KUKA KRL program: EPS_2_25990_SANMH02_A_20260122125454.src

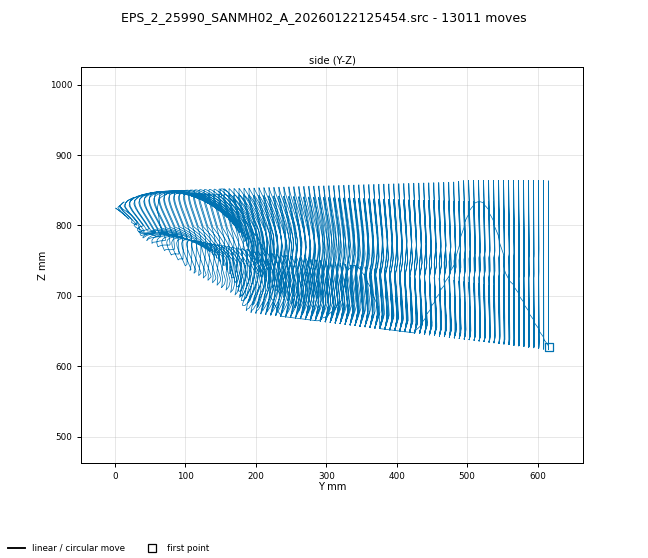
[picture p0: tool path of EPS_2_25990_SANMH02_A_20260122125454.src, 13011 of 13013 moves have a stored position in this frame; points joined in program order, loops and branches not executed]
&ACCESS RVP
&REL 4
&COMMENT QRS 19112012
&PARAM EDITMASK = *
DEF PART()
EXT BAS (BAS_COMMAND :IN,REAL :IN )
INT I
BAS (#INITMOV,0 )

;KUKA QRS Post kuka4.cps  Date:22-06-2017 !

File_ID=3005

QRS_PRE_INIT()

;Init var - Until changes are made in qrs_pre_init
Outlet_Square_prg=0
Inlet_1_Square_prg=0
Inlet_2_Square_prg=0
Inlet_3_Square_prg=0
Inlet_4_Square_prg=0
Inlet_5_Square_prg=0

Outlet_1={X 0.000, Y 498.690, Z 763.500, B 0.000, E1 0.000 }
Inlet_1={X 0.000, Y 500.880, Z 733.500, B 0.000, E1 131.000 }
Inlet_2={X 0.000, Y 537.160, Z 233.500, B 0.000, E1 218.000 }
Outlet_1_type=201
Inlet_1_type=201
Inlet_2_type=201
;QRS#1=Sidecore dimensions
;QRS#2=200-8" PVC SDR 35
;QRS#3=200-8" PVC SDR 35
;QRS#4=200-8" PVC SDR 35
;QRS#5=
;QRS#6=
;QRS#7=
;QRS#8=
;QRS#9=12-08 PSX
;QRS#10=12-08 PSX
;QRS#11=12-08 PSX
;QRS#12=
;QRS#13=
;QRS#14=
;QRS#15=
;QRS#16=1220x127x1143 3,75'
;QRS#17=EPS Height
;QRS#18=864
;QRS#19=*
;QRS#20= UPDATED VERSION 22-06-2017
;QRS#21=*
Outlet_Square=0100
Inlet_1_Square=0100
Inlet_2_Square=0100
Inlet_3_Square=0
Inlet_4_Square=0
Inlet_5_Square=0
Mill_Square=1
Outlet_Square_Prg=204
Inlet_1_Square_prg=204
Inlet_2_Square_prg=204

QRS_INIT()

$ADVANCE=5

; T1
PTP {E1 173.412,E2 173.412}
PTP {X 0,Y 615.492,A -85,B 0,C 180,E1 173.412,E2 173.412,E3 0,E4 0,E5 0,E6 0}
QRS_SPEED_INIT()
LIN {X 0,Y 615.492,Z 627.912,A -85,B 0,C 180,E1 173.412,E2 173.412,E3 0,E4 0,E5 0,E6 0} C_VEL
LIN {X 0,Y 615.475,Z 638.168,A -85,B 0,C 180,E1 170.801,E2 170.801} C_VEL
LIN {X 0,Y 615.49,Z 648.911,A -85,B 0,C 180,E1 168.139,E2 168.139} C_VEL
LIN {X 0,Y 615.487,Z 660.046,A -85,B 0,C 180,E1 165.451,E2 165.451} C_VEL
LIN {X 0,Y 615.476,Z 671.583,A -85,B 0,C 180,E1 162.729,E2 162.729} C_VEL
LIN {X 0,Y 615.485,Z 683.521,A -85,B 0,C 180,E1 159.967,E2 159.967} C_VEL
LIN {X 0,Y 615.487,Z 695.908,A -85,B 0,C 180,E1 157.155,E2 157.155} C_VEL
LIN {X 0,Y 615.494,Z 708.733,A -85,B 0,C 180,E1 154.285,E2 154.285} C_VEL
LIN {X 0,Y 615.476,Z 721.128,A -85,B 0,C 180,E1 151.55,E2 151.55} C_VEL
LIN {X 0,Y 615.494,Z 725.535,A -85,B 0,C 180,E1 150.606,E2 150.606} C_VEL
LIN {X 0,Y 615.488,Z 739.328,A -85,B 0,C 180,E1 150.351,E2 150.351} C_VEL
LIN {X 0,Y 615.49,Z 751.99,A -85,B 0,C 180,E1 149.977,E2 149.977} C_VEL
LIN {X 0,Y 615.476,Z 764.482,A -85,B 0,C 180,E1 149.46,E2 149.46} C_VEL
LIN {X 0,Y 615.493,Z 776.033,A -85,B 0,C 180,E1 148.838,E2 148.838} C_VEL
LIN {X 0,Y 615.5,Z 786.168,A -85,B 0,C 180,E1 148.154,E2 148.154} C_VEL
LIN {X 0,Y 615.499,Z 795.798,A -85,B 0,C 180,E1 147.349,E2 147.349} C_VEL
LIN {X 0,Y 615.496,Z 804.466,A -85,B 0,C 180,E1 146.463,E2 146.463} C_VEL
LIN {X 0,Y 615.497,Z 812.382,A -85,B 0,C 180,E1 145.468,E2 145.468} C_VEL
LIN {X 0,Y 615.496,Z 819.171,A -85,B 0,C 180,E1 144.385,E2 144.385} C_VEL
LIN {X 0,Y 615.496,Z 824.387,A -85,B 0,C 180,E1 143.319,E2 143.319} C_VEL
LIN {X 0,Y 615.497,Z 827.932,A -85,B 0,C 180,E1 142.373,E2 142.373} C_VEL
LIN {X 0,Y 615.498,Z 831.277,A -85,B 0,C 180,E1 141.096,E2 141.096} C_VEL
LIN {X 0,Y 615.495,Z 832.963,A -85,B 0,C 180,E1 139.909,E2 139.909} C_VEL
LIN {X 0,Y 615.492,Z 833.383,A -85,B 0,C 180,E1 138.904,E2 138.904} C_VEL
LIN {X 0,Y 615.498,Z 832.581,A -85,B 0,C 180,E1 137.648,E2 137.648} C_VEL
LIN {X 0,Y 615.499,Z 831.153,A -85,B 0,C 180,E1 136.756,E2 136.756} C_VEL
LIN {X 0,Y 615.496,Z 827.689,A -85,B 0,C 180,E1 135.46,E2 135.46} C_VEL
LIN {X 0,Y 615.495,Z 824.163,A -85,B 0,C 180,E1 134.539,E2 134.539} C_VEL
LIN {X 0,Y 615.497,Z 818.654,A -85,B 0,C 180,E1 133.431,E2 133.431} C_VEL
LIN {X 0,Y 615.495,Z 811.719,A -85,B 0,C 180,E1 132.352,E2 132.352} C_VEL
LIN {X 0,Y 615.494,Z 803.005,A -85,B 0,C 180,E1 131.284,E2 131.284} C_VEL
LIN {X 0,Y 615.498,Z 794.891,A -85,B 0,C 180,E1 130.476,E2 130.476} C_VEL
LIN {X 0,Y 615.497,Z 784.864,A -85,B 0,C 180,E1 129.662,E2 129.662} C_VEL
LIN {X 0,Y 615.487,Z 773.182,A -85,B 0,C 180,E1 128.904,E2 128.904} C_VEL
LIN {X 0,Y 615.479,Z 761.912,A -85,B 0,C 180,E1 128.328,E2 128.328} C_VEL
LIN {X 0,Y 615.483,Z 749.983,A -85,B 0,C 180,E1 127.866,E2 127.866} C_VEL
LIN {X 0,Y 615.496,Z 736.899,A -85,B 0,C 180,E1 127.504,E2 127.504} C_VEL
LIN {X 0,Y 615.489,Z 725.354,A -85,B 0,C 180,E1 127.289,E2 127.289} C_VEL
LIN {X 0,Y 615.49,Z 713.598,A -85,B 0,C 180,E1 124.701,E2 124.701} C_VEL
LIN {X 0,Y 615.481,Z 701.48,A -85,B 0,C 180,E1 122.007,E2 122.007} C_VEL
LIN {X 0,Y 615.493,Z 689.933,A -85,B 0,C 180,E1 119.405,E2 119.405} C_VEL
LIN {X 0,Y 615.476,Z 678.313,A -85,B 0,C 180,E1 116.743,E2 116.743} C_VEL
LIN {X 0,Y 615.488,Z 666.578,A -85,B 0,C 180,E1 114.008,E2 114.008} C_VEL
LIN {X 0,Y 615.492,Z 655.757,A -85,B 0,C 180,E1 111.431,E2 111.431} C_VEL
LIN {X 0,Y 615.48,Z 644.161,A -85,B 0,C 180,E1 108.603,E2 108.603} C_VEL
LIN {X 0,Y 615.484,Z 633.399,A -85,B 0,C 180,E1 105.905,E2 105.905} C_VEL
LIN {X 0,Y 615.488,Z 623.694,A -85,B 0,C 180,E1 103.369,E2 103.369} C_VEL
LIN {X 0,Y 615.476,Z 623.696,A -85,B 0,C 180,E1 100.527,E2 100.527} C_VEL
LIN {X 0,Y 615.484,Z 623.694,A -85,B 0,C 180,E1 97.875,E2 97.875} C_VEL
LIN {X 0,Y 615.485,Z 623.694,A -85,B 0,C 180,E1 95.241,E2 95.241} C_VEL
LIN {X 0,Y 615.477,Z 623.696,A -85,B 0,C 180,E1 92.618,E2 92.618} C_VEL
LIN {X 0,Y 615.491,Z 623.693,A -85,B 0,C 180,E1 90,E2 90} C_VEL
LIN {X 0,Y 615.477,Z 623.696,A -85,B 0,C 180,E1 87.382,E2 87.382} C_VEL
LIN {X 0,Y 615.485,Z 623.695,A -85,B 0,C 180,E1 84.758,E2 84.758} C_VEL
LIN {X 0,Y 615.488,Z 623.694,A -85,B 0,C 180,E1 82.124,E2 82.124} C_VEL
LIN {X 0,Y 615.477,Z 623.697,A -85,B 0,C 180,E1 79.473,E2 79.473} C_VEL
LIN {X 0,Y 615.497,Z 623.692,A -85,B 0,C 180,E1 76.799,E2 76.799} C_VEL
LIN {X 0,Y 615.481,Z 623.695,A -85,B 0,C 180,E1 74.094,E2 74.094} C_VEL
LIN {X 0,Y 615.477,Z 623.696,A -85,B 0,C 180,E1 71.353,E2 71.353} C_VEL
LIN {X 0,Y 615.492,Z 623.693,A -85,B 0,C 180,E1 68.568,E2 68.568} C_VEL
LIN {X 0,Y 615.489,Z 623.695,A -85,B 0,C 180,E1 65.728,E2 65.728} C_VEL
LIN {X 0,Y 615.482,Z 623.695,A -85,B 0,C 180,E1 63.237,E2 63.237} C_VEL
LIN {X 0,Y 615.484,Z 636.143,A -85,B 0,C 180,E1 62.823,E2 62.823} C_VEL
LIN {X 0,Y 615.481,Z 648.35,A -85,B 0,C 180,E1 62.269,E2 62.269} C_VEL
LIN {X 0,Y 615.492,Z 659.541,A -85,B 0,C 180,E1 61.615,E2 61.615} C_VEL
LIN {X 0,Y 615.5,Z 669.72,A -85,B 0,C 180,E1 60.875,E2 60.875} C_VEL
LIN {X 0,Y 615.498,Z 679.215,A -85,B 0,C 180,E1 60.022,E2 60.022} C_VEL
LIN {X 0,Y 615.497,Z 687.701,A -85,B 0,C 180,E1 59.081,E2 59.081} C_VEL
LIN {X 0,Y 615.498,Z 694.509,A -85,B 0,C 180,E1 58.154,E2 58.154} C_VEL
LIN {X 0,Y 615.495,Z 700.434,A -85,B 0,C 180,E1 57.154,E2 57.154} C_VEL
LIN {X 0,Y 615.495,Z 705.787,A -85,B 0,C 180,E1 55.978,E2 55.978} C_VEL
LIN {X 0,Y 615.497,Z 709.663,A -85,B 0,C 180,E1 54.786,E2 54.786} C_VEL
LIN {X 0,Y 615.495,Z 712.179,A -85,B 0,C 180,E1 53.576,E2 53.576} C_VEL
LIN {X 0,Y 615.495,Z 713.068,A -85,B 0,C 180,E1 52.758,E2 52.758} C_VEL
LIN {X 0,Y 615.494,Z 713.388,A -85,B 0,C 180,E1 51.932,E2 51.932} C_VEL
LIN {X 0,Y 615.495,Z 712.915,A -85,B 0,C 180,E1 50.937,E2 50.937} C_VEL
LIN {X 0,Y 615.496,Z 711.471,A -85,B 0,C 180,E1 49.91,E2 49.91} C_VEL
LIN {X 0,Y 615.494,Z 709.077,A -85,B 0,C 180,E1 48.905,E2 48.905} C_VEL
LIN {X 0,Y 615.497,Z 705.739,A -85,B 0,C 180,E1 47.919,E2 47.919} C_VEL
LIN {X 0,Y 615.498,Z 700.437,A -85,B 0,C 180,E1 46.756,E2 46.756} C_VEL
LIN {X 0,Y 615.494,Z 693.832,A -85,B 0,C 180,E1 45.656,E2 45.656} C_VEL
LIN {X 0,Y 615.495,Z 686.933,A -85,B 0,C 180,E1 44.735,E2 44.735} C_VEL
LIN {X 0,Y 615.498,Z 678.433,A -85,B 0,C 180,E1 43.808,E2 43.808} C_VEL
LIN {X 0,Y 615.499,Z 668.778,A -85,B 0,C 180,E1 42.961,E2 42.961} C_VEL
LIN {X 0,Y 615.492,Z 658.341,A -85,B 0,C 180,E1 42.216,E2 42.216} C_VEL
LIN {X 0,Y 615.476,Z 648.077,A -85,B 0,C 180,E1 41.626,E2 41.626} C_VEL
LIN {X 0,Y 615.488,Z 636.331,A -85,B 0,C 180,E1 41.095,E2 41.095} C_VEL
LIN {X 0,Y 615.492,Z 623.695,A -85,B 0,C 180,E1 40.667,E2 40.667} C_VEL
LIN {X 0,Y 615.488,Z 623.688,A -85,B 0,C 180,E1 38.012,E2 38.012} C_VEL
LIN {X 0,Y 615.476,Z 623.685,A -85,B 0,C 180,E1 35.617,E2 35.617} C_VEL
LIN {X 0,Y 615.48,Z 623.683,A -85,B 0,C 180,E1 33.237,E2 33.237} C_VEL
LIN {X 0,Y 615.489,Z 623.685,A -85,B 0,C 180,E1 30.92,E2 30.92} C_VEL
LIN {X 0,Y 615.494,Z 623.697,A -85,B 0,C 180,E1 28.451,E2 28.451} C_VEL
LIN {X 0,Y 615.478,Z 623.685,A -85,B 0,C 180,E1 25.567,E2 25.567} C_VEL
LIN {X 0,Y 615.489,Z 623.684,A -85,B 0,C 180,E1 22.844,E2 22.844} C_VEL
LIN {X 0,Y 615.493,Z 623.695,A -85,B 0,C 180,E1 20.033,E2 20.033} C_VEL
LIN {X 0,Y 615.476,Z 623.684,A -85,B 0,C 180,E1 17.271,E2 17.271} C_VEL
LIN {X 0,Y 615.489,Z 623.688,A -85,B 0,C 180,E1 14.549,E2 14.549} C_VEL
LIN {X 0,Y 615.49,Z 623.693,A -85,B 0,C 180,E1 11.861,E2 11.861} C_VEL
LIN {X 0,Y 615.475,Z 623.684,A -85,B 0,C 180,E1 9.199,E2 9.199} C_VEL
LIN {X 0,Y 615.492,Z 623.685,A -85,B 0,C 180,E1 6.557,E2 6.557} C_VEL
LIN {X 0,Y 615.489,Z 623.7,A -85,B 0,C 180,E1 3.928,E2 3.928} C_VEL
LIN {X 0,Y 615.484,Z 623.685,A -85,B 0,C 180,E1 1.308,E2 1.308} C_VEL
LIN {X 0,Y 615.484,Z 623.683,A -85,B 0,C 180,E1 -1.309,E2 -1.309} C_VEL
LIN {X 0,Y 615.493,Z 623.694,A -85,B 0,C 180,E1 -3.929,E2 -3.929} C_VEL
LIN {X 0,Y 615.487,Z 623.689,A -85,B 0,C 180,E1 -6.579,E2 -6.579} C_VEL
LIN {X 0,Y 615.475,Z 623.684,A -85,B 0,C 180,E1 -9.199,E2 -9.199} C_VEL
LIN {X 0,Y 615.494,Z 623.688,A -85,B 0,C 180,E1 -11.861,E2 -11.861} C_VEL
LIN {X 0,Y 615.483,Z 623.694,A -85,B 0,C 180,E1 -14.549,E2 -14.549} C_VEL
LIN {X 0,Y 615.476,Z 623.684,A -85,B 0,C 180,E1 -17.271,E2 -17.271} C_VEL
LIN {X 0,Y 615.494,Z 623.69,A -85,B 0,C 180,E1 -20.033,E2 -20.033} C_VEL
LIN {X 0,Y 615.486,Z 623.688,A -85,B 0,C 180,E1 -22.845,E2 -22.845} C_VEL
LIN {X 0,Y 615.478,Z 623.684,A -85,B 0,C 180,E1 -25.567,E2 -25.567} C_VEL
LIN {X 0,Y 615.497,Z 623.7,A -85,B 0,C 180,E1 -28.452,E2 -28.452} C_VEL
LIN {X 0,Y 615.483,Z 623.686,A -85,B 0,C 180,E1 -31.085,E2 -31.085} C_VEL
LIN {X 0,Y 615.476,Z 623.684,A -85,B 0,C 180,E1 -33.533,E2 -33.533} C_VEL
LIN {X 0,Y 615.488,Z 623.697,A -85,B 0,C 180,E1 -36.425,E2 -36.425} C_VEL
LIN {X 0,Y 615.492,Z 623.687,A -85,B 0,C 180,E1 -39.063,E2 -39.063} C_VEL
LIN {X 0,Y 615.481,Z 623.683,A -85,B 0,C 180,E1 -41.475,E2 -41.475} C_VEL
LIN {X 0,Y 615.493,Z 623.685,A -85,B 0,C 180,E1 -44.149,E2 -44.149} C_VEL
LIN {X 0,Y 615.486,Z 623.695,A -85,B 0,C 180,E1 -46.953,E2 -46.953} C_VEL
LIN {X 0,Y 615.483,Z 623.685,A -85,B 0,C 180,E1 -49.393,E2 -49.393} C_VEL
LIN {X 0,Y 615.477,Z 623.684,A -85,B 0,C 180,E1 -51.99,E2 -51.99} C_VEL
LIN {X 0,Y 615.496,Z 623.801,A -85,B 0,C 180,E1 -54.358,E2 -54.358} C_VEL
LIN {X 0,Y 615.48,Z 637.627,A -85,B 0,C 180,E1 -57.153,E2 -57.153} C_VEL
LIN {X 0,Y 615.488,Z 651.322,A -85,B 0,C 180,E1 -59.84,E2 -59.84} C_VEL
LIN {X 0,Y 615.487,Z 665.016,A -85,B 0,C 180,E1 -62.454,E2 -62.454} C_VEL
LIN {X 0,Y 615.481,Z 680.66,A -85,B 0,C 180,E1 -65.368,E2 -65.368} C_VEL
LIN {X 0,Y 615.477,Z 696.292,A -85,B 0,C 180,E1 -68.216,E2 -68.216} C_VEL
LIN {X 0,Y 615.481,Z 711.904,A -85,B 0,C 180,E1 -71.008,E2 -71.008} C_VEL
LIN {X 0,Y 615.494,Z 727.95,A -85,B 0,C 180,E1 -73.833,E2 -73.833} C_VEL
LIN {X 0,Y 615.498,Z 745.032,A -85,B 0,C 180,E1 -76.799,E2 -76.799} C_VEL
LIN {X 0,Y 615.475,Z 753.922,A -85,B 0,C 180,E1 -78.327,E2 -78.327} C_VEL
LIN {X 0,Y 615.481,Z 767.23,A -85,B 0,C 180,E1 -78.556,E2 -78.556} C_VEL
LIN {X 0,Y 615.492,Z 780.365,A -85,B 0,C 180,E1 -78.923,E2 -78.923} C_VEL
LIN {X 0,Y 615.475,Z 792.144,A -85,B 0,C 180,E1 -79.384,E2 -79.384} C_VEL
LIN {X 0,Y 615.489,Z 803.57,A -85,B 0,C 180,E1 -79.972,E2 -79.972} C_VEL
LIN {X 0,Y 615.499,Z 815.017,A -85,B 0,C 180,E1 -80.718,E2 -80.718} C_VEL
LIN {X 0,Y 615.498,Z 824.254,A -85,B 0,C 180,E1 -81.463,E2 -81.463} C_VEL
LIN {X 0,Y 615.499,Z 832.651,A -85,B 0,C 180,E1 -82.289,E2 -82.289} C_VEL
LIN {X 0,Y 615.497,Z 840.69,A -85,B 0,C 180,E1 -83.259,E2 -83.259} C_VEL
LIN {X 0,Y 615.498,Z 846.421,A -85,B 0,C 180,E1 -84.101,E2 -84.101} C_VEL
LIN {X 0,Y 615.497,Z 851.871,A -85,B 0,C 180,E1 -85.087,E2 -85.087} C_VEL
LIN {X 0,Y 615.497,Z 856.14,A -85,B 0,C 180,E1 -86.071,E2 -86.071} C_VEL
LIN {X 0,Y 615.496,Z 858.397,A -85,B 0,C 180,E1 -86.727,E2 -86.727} C_VEL
LIN {X 0,Y 615.497,Z 860.232,A -85,B 0,C 180,E1 -87.382,E2 -87.382} C_VEL
LIN {X 0,Y 615.496,Z 861.608,A -85,B 0,C 180,E1 -88.037,E2 -88.037} C_VEL
LIN {X 0,Y 615.496,Z 863.173,A -85,B 0,C 180,E1 -89.345,E2 -89.345} C_VEL
LIN {X 0,Y 615.494,Z 863.389,A -85,B 0,C 180,E1 -90,E2 -90} C_VEL
LIN {X 0,Y 615.496,Z 862.58,A -85,B 0,C 180,E1 -91.308,E2 -91.308} C_VEL
LIN {X 0,Y 615.496,Z 861.609,A -85,B 0,C 180,E1 -91.963,E2 -91.963} C_VEL
LIN {X 0,Y 615.497,Z 860.234,A -85,B 0,C 180,E1 -92.617,E2 -92.617} C_VEL
LIN {X 0,Y 615.496,Z 857.351,A -85,B 0,C 180,E1 -93.6,E2 -93.6} C_VEL
LIN {X 0,Y 615.498,Z 853.443,A -85,B 0,C 180,E1 -94.584,E2 -94.584} C_VEL
LIN {X 0,Y 615.499,Z 848.407,A -85,B 0,C 180,E1 -95.569,E2 -95.569} C_VEL
LIN {X 0,Y 615.497,Z 841.87,A -85,B 0,C 180,E1 -96.583,E2 -96.583} C_VEL
LIN {X 0,Y 615.497,Z 834.137,A -85,B 0,C 180,E1 -97.545,E2 -97.545} C_VEL
LIN {X 0,Y 615.498,Z 826.049,A -85,B 0,C 180,E1 -98.371,E2 -98.371} C_VEL
LIN {X 0,Y 615.499,Z 816.173,A -85,B 0,C 180,E1 -99.198,E2 -99.198} C_VEL
LIN {X 0,Y 615.484,Z 804.989,A -85,B 0,C 180,E1 -99.945,E2 -99.945} C_VEL
LIN {X 0,Y 615.476,Z 794.033,A -85,B 0,C 180,E1 -100.527,E2 -100.527} C_VEL
LIN {X 0,Y 615.489,Z 781.554,A -85,B 0,C 180,E1 -101.038,E2 -101.038} C_VEL
LIN {X 0,Y 615.483,Z 769.085,A -85,B 0,C 180,E1 -101.401,E2 -101.401} C_VEL
LIN {X 0,Y 615.475,Z 755.501,A -85,B 0,C 180,E1 -101.652,E2 -101.652} C_VEL
LIN {X 0,Y 615.475,Z 753.8,A -85,B 0,C 180,E1 -101.693,E2 -101.693} C_VEL
LIN {X 0,Y 615.491,Z 739.038,A -85,B 0,C 180,E1 -104.238,E2 -104.238} C_VEL
LIN {X 0,Y 615.477,Z 723.612,A -85,B 0,C 180,E1 -106.928,E2 -106.928} C_VEL
LIN {X 0,Y 615.491,Z 709.955,A -85,B 0,C 180,E1 -109.337,E2 -109.337} C_VEL
LIN {X 0,Y 615.479,Z 694.341,A -85,B 0,C 180,E1 -112.136,E2 -112.136} C_VEL
LIN {X 0,Y 615.481,Z 680.664,A -85,B 0,C 180,E1 -114.631,E2 -114.631} C_VEL
LIN {X 0,Y 615.491,Z 665.021,A -85,B 0,C 180,E1 -117.545,E2 -117.545} C_VEL
LIN {X 0,Y 615.485,Z 651.326,A -85,B 0,C 180,E1 -120.16,E2 -120.16} C_VEL
LIN {X 0,Y 615.48,Z 637.631,A -85,B 0,C 180,E1 -122.846,E2 -122.846} C_VEL
LIN {X 0,Y 615.494,Z 623.687,A -85,B 0,C 180,E1 -125.669,E2 -125.669} C_VEL
LIN {X 0,Y 615.476,Z 623.686,A -85,B 0,C 180,E1 -128.069,E2 -128.069} C_VEL
LIN {X 0,Y 615.487,Z 623.694,A -85,B 0,C 180,E1 -130.606,E2 -130.606} C_VEL
LIN {X 0,Y 615.478,Z 623.69,A -85,B 0,C 180,E1 -133.245,E2 -133.245} C_VEL
LIN {X 0,Y 615.488,Z 623.687,A -85,B 0,C 180,E1 -136.002,E2 -136.002} C_VEL
LIN {X 0,Y 615.484,Z 623.69,A -85,B 0,C 180,E1 -138.905,E2 -138.905} C_VEL
LIN {X 0,Y 615.482,Z 623.686,A -85,B 0,C 180,E1 -141.095,E2 -141.095} C_VEL
LIN {X 0,Y 615.479,Z 623.689,A -85,B 0,C 180,E1 -143.574,E2 -143.574} C_VEL
LIN {X 0,Y 615.476,Z 623.693,A -85,B 0,C 180,E1 -146.466,E2 -146.466} C_VEL
LIN {X 0,Y 615.485,Z 623.685,A -85,B 0,C 180,E1 -149.08,E2 -149.08} C_VEL
LIN {X 0,Y 615.476,Z 623.698,A -85,B 0,C 180,E1 -151.55,E2 -151.55} C_VEL
LIN {X 0,Y 615.484,Z 623.687,A -85,B 0,C 180,E1 -154.284,E2 -154.284} C_VEL
LIN {X 0,Y 615.479,Z 623.686,A -85,B 0,C 180,E1 -156.443,E2 -156.443} C_VEL
LIN {X 0,Y 615.493,Z 623.699,A -85,B 0,C 180,E1 -159.269,E2 -159.269} C_VEL
LIN {X 0,Y 615.488,Z 623.684,A -85,B 0,C 180,E1 -162.043,E2 -162.043} C_VEL
LIN {X 0,Y 615.486,Z 623.694,A -85,B 0,C 180,E1 -164.774,E2 -164.774} C_VEL
LIN {X 0,Y 615.486,Z 623.688,A -85,B 0,C 180,E1 -167.47,E2 -167.47} C_VEL
LIN {X 0,Y 615.485,Z 623.687,A -85,B 0,C 180,E1 -170.138,E2 -170.138} C_VEL
LIN {X 0,Y 615.481,Z 623.699,A -85,B 0,C 180,E1 -172.784,E2 -172.784} C_VEL
LIN {X 0,Y 615.497,Z 623.682,A -85,B 0,C 180,E1 -175.415,E2 -175.415} C_VEL
LIN {X 0,Y 615.476,Z 623.695,A -85,B 0,C 180,E1 -178.037,E2 -178.037} C_VEL
LIN {X 0,Y 615.483,Z 623.691,A -85,B 0,C 180,E1 -180.654,E2 -180.654} C_VEL
LIN {X 0,Y 615.481,Z 623.686,A -85,B 0,C 180,E1 -183.273,E2 -183.273} C_VEL
LIN {X 0,Y 615.494,Z 623.838,A -85,B 0,C 180,E1 -185.529,E2 -185.529} C_VEL
LIN {X 0,Y 615.492,Z 627.912,A -85,B 0,C 180,E1 -186.588,E2 -186.588} C_VEL
LIN {X 0,Y 614.818,Z 630.052,A -85,B 0,C 180,E1 -187.098,E2 -187.098} C_VEL
LIN {X 0,Y 609.193,Z 637.77,A -85,B 0,C 180,E1 -188.729,E2 -188.729} C_VEL
LIN {X 0,Y 608.556,Z 639.946,A -85,B 0,C 180,E1 -189.245,E2 -189.245} C_VEL
LIN {X 0,Y 608.537,Z 650.962,A -85,B 0,C 180,E1 -191.998,E2 -191.998} C_VEL
LIN {X 0,Y 608.507,Z 662.145,A -85,B 0,C 180,E1 -194.72,E2 -194.72} C_VEL
LIN {X 0,Y 608.494,Z 673.735,A -85,B 0,C 180,E1 -197.475,E2 -197.475} C_VEL
LIN {X 0,Y 608.486,Z 684.228,A -85,B 0,C 180,E1 -199.921,E2 -199.921} C_VEL
LIN {X 0,Y 608.453,Z 695.382,A -85,B 0,C 180,E1 -202.477,E2 -202.477} C_VEL
LIN {X 0,Y 608.475,Z 706.26,A -85,B 0,C 180,E1 -204.934,E2 -204.934} C_VEL
LIN {X 0,Y 608.455,Z 719.53,A -85,B 0,C 180,E1 -207.891,E2 -207.891} C_VEL
LIN {X 0,Y 608.444,Z 725.728,A -85,B 0,C 180,E1 -209.258,E2 -209.258} C_VEL
LIN {X 0,Y 608.53,Z 739.322,A -85,B 0,C 180,E1 -209.514,E2 -209.514} C_VEL
LIN {X 0,Y 608.541,Z 752.298,A -85,B 0,C 180,E1 -209.902,E2 -209.902} C_VEL
LIN {X 0,Y 608.49,Z 763.922,A -85,B 0,C 180,E1 -210.384,E2 -210.384} C_VEL
LIN {X 0,Y 608.485,Z 775.86,A -85,B 0,C 180,E1 -211.025,E2 -211.025} C_VEL
LIN {X 0,Y 608.497,Z 785.904,A -85,B 0,C 180,E1 -211.703,E2 -211.703} C_VEL
LIN {X 0,Y 608.469,Z 795.789,A -85,B 0,C 180,E1 -212.525,E2 -212.525} C_VEL
LIN {X 0,Y 608.474,Z 805.008,A -85,B 0,C 180,E1 -213.471,E2 -213.471} C_VEL
LIN {X 0,Y 608.463,Z 812.881,A -85,B 0,C 180,E1 -214.47,E2 -214.47} C_VEL
LIN {X 0,Y 608.446,Z 819.187,A -85,B 0,C 180,E1 -215.469,E2 -215.469} C_VEL
LIN {X 0,Y 608.453,Z 824.357,A -85,B 0,C 180,E1 -216.502,E2 -216.502} C_VEL
LIN {X 0,Y 608.435,Z 829.002,A -85,B 0,C 180,E1 -217.749,E2 -217.749} C_VEL
LIN {X 0,Y 608.428,Z 831.244,A -85,B 0,C 180,E1 -218.591,E2 -218.591} C_VEL
LIN {X 0,Y 608.421,Z 832.839,A -85,B 0,C 180,E1 -219.443,E2 -219.443} C_VEL
LIN {X 0,Y 608.427,Z 833.744,A -85,B 0,C 180,E1 -220.327,E2 -220.327} C_VEL
LIN {X 0,Y 608.42,Z 833.937,A -85,B 0,C 180,E1 -221.339,E2 -221.339} C_VEL
LIN {X 0,Y 608.438,Z 833.226,A -85,B 0,C 180,E1 -222.333,E2 -222.333} C_VEL
LIN {X 0,Y 608.435,Z 831.66,A -85,B 0,C 180,E1 -223.306,E2 -223.306} C_VEL
LIN {X 0,Y 608.424,Z 829.257,A -85,B 0,C 180,E1 -224.262,E2 -224.262} C_VEL
LIN {X 0,Y 608.437,Z 824.745,A -85,B 0,C 180,E1 -225.497,E2 -225.497} C_VEL
LIN {X 0,Y 608.437,Z 818.782,A -85,B 0,C 180,E1 -226.695,E2 -226.695} C_VEL
LIN {X 0,Y 608.468,Z 811.538,A -85,B 0,C 180,E1 -227.804,E2 -227.804} C_VEL
LIN {X 0,Y 608.451,Z 803.18,A -85,B 0,C 180,E1 -228.824,E2 -228.824} C_VEL
LIN {X 0,Y 608.464,Z 794.334,A -85,B 0,C 180,E1 -229.698,E2 -229.698} C_VEL
LIN {X 0,Y 608.48,Z 783.487,A -85,B 0,C 180,E1 -230.562,E2 -230.562} C_VEL
LIN {X 0,Y 608.492,Z 773.541,A -85,B 0,C 180,E1 -231.203,E2 -231.203} C_VEL
LIN {X 0,Y 608.492,Z 761.414,A -85,B 0,C 180,E1 -231.823,E2 -231.823} C_VEL
LIN {X 0,Y 608.532,Z 748.966,A -85,B 0,C 180,E1 -232.3,E2 -232.3} C_VEL
LIN {X 0,Y 608.539,Z 736.298,A -85,B 0,C 180,E1 -232.645,E2 -232.645} C_VEL
LIN {X 0,Y 608.436,Z 725.658,A -85,B 0,C 180,E1 -232.846,E2 -232.846} C_VEL
LIN {X 0,Y 608.451,Z 713.533,A -85,B 0,C 180,E1 -235.53,E2 -235.53} C_VEL
LIN {X 0,Y 608.471,Z 701.192,A -85,B 0,C 180,E1 -238.296,E2 -238.296} C_VEL
LIN {X 0,Y 608.473,Z 689.39,A -85,B 0,C 180,E1 -240.981,E2 -240.981} C_VEL
LIN {X 0,Y 608.515,Z 678.064,A -85,B 0,C 180,E1 -243.6,E2 -243.6} C_VEL
LIN {X 0,Y 608.503,Z 665.7,A -85,B 0,C 180,E1 -246.518,E2 -246.518} C_VEL
LIN {X 0,Y 608.536,Z 655.323,A -85,B 0,C 180,E1 -249.022,E2 -249.022} C_VEL
LIN {X 0,Y 608.557,Z 643.961,A -85,B 0,C 180,E1 -251.832,E2 -251.832} C_VEL
LIN {X 0,Y 608.585,Z 633.096,A -85,B 0,C 180,E1 -254.598,E2 -254.598} C_VEL
LIN {X 0,Y 608.556,Z 626.367,A -85,B 0,C 180,E1 -256.306,E2 -256.306} C_VEL
LIN {X 0,Y 608.465,Z 624.693,A -85,B 0,C 180,E1 -256.729,E2 -256.729} C_VEL
LIN {X 0,Y 608.457,Z 624.693,A -85,B 0,C 180,E1 -259.35,E2 -259.35} C_VEL
LIN {X 0,Y 608.477,Z 624.69,A -85,B 0,C 180,E1 -262.033,E2 -262.033} C_VEL
LIN {X 0,Y 608.466,Z 624.692,A -85,B 0,C 180,E1 -264.699,E2 -264.699} C_VEL
LIN {X 0,Y 608.469,Z 624.691,A -85,B 0,C 180,E1 -267.352,E2 -267.352} C_VEL
LIN {X 0,Y 608.481,Z 624.69,A -85,B 0,C 180,E1 -270,E2 -270} C_VEL
LIN {X 0,Y 608.469,Z 624.691,A -85,B 0,C 180,E1 -272.648,E2 -272.648} C_VEL
LIN {X 0,Y 608.464,Z 624.692,A -85,B 0,C 180,E1 -275.302,E2 -275.302} C_VEL
LIN {X 0,Y 608.481,Z 624.69,A -85,B 0,C 180,E1 -277.967,E2 -277.967} C_VEL
LIN {X 0,Y 608.457,Z 624.693,A -85,B 0,C 180,E1 -280.65,E2 -280.65} C_VEL
LIN {X 0,Y 608.472,Z 624.691,A -85,B 0,C 180,E1 -283.356,E2 -283.356} C_VEL
LIN {X 0,Y 608.461,Z 624.692,A -85,B 0,C 180,E1 -286.094,E2 -286.094} C_VEL
LIN {X 0,Y 608.453,Z 624.694,A -85,B 0,C 180,E1 -288.87,E2 -288.87} C_VEL
LIN {X 0,Y 608.476,Z 624.692,A -85,B 0,C 180,E1 -291.691,E2 -291.691} C_VEL
LIN {X 0,Y 608.452,Z 624.698,A -85,B 0,C 180,E1 -294.571,E2 -294.571} C_VEL
LIN {X 0,Y 608.473,Z 624.728,A -85,B 0,C 180,E1 -296.658,E2 -296.658} C_VEL
LIN {X 0,Y 608.503,Z 636.887,A -85,B 0,C 180,E1 -297.076,E2 -297.076} C_VEL
LIN {X 0,Y 608.486,Z 648.492,A -85,B 0,C 180,E1 -297.61,E2 -297.61} C_VEL
LIN {X 0,Y 608.477,Z 659.647,A -85,B 0,C 180,E1 -298.266,E2 -298.266} C_VEL
LIN {X 0,Y 608.486,Z 669.952,A -85,B 0,C 180,E1 -299.019,E2 -299.019} C_VEL
LIN {X 0,Y 608.483,Z 678.482,A -85,B 0,C 180,E1 -299.779,E2 -299.779} C_VEL
LIN {X 0,Y 608.46,Z 687.169,A -85,B 0,C 180,E1 -300.726,E2 -300.726} C_VEL
LIN {X 0,Y 608.463,Z 694.464,A -85,B 0,C 180,E1 -301.705,E2 -301.705} C_VEL
LIN {X 0,Y 608.433,Z 699.452,A -85,B 0,C 180,E1 -302.518,E2 -302.518} C_VEL
LIN {X 0,Y 608.425,Z 705.322,A -85,B 0,C 180,E1 -303.728,E2 -303.728} C_VEL
LIN {X 0,Y 608.424,Z 709.484,A -85,B 0,C 180,E1 -304.902,E2 -304.902} C_VEL
LIN {X 0,Y 608.423,Z 712.259,A -85,B 0,C 180,E1 -306.094,E2 -306.094} C_VEL
LIN {X 0,Y 608.434,Z 713.622,A -85,B 0,C 180,E1 -307.154,E2 -307.154} C_VEL
LIN {X 0,Y 608.42,Z 713.962,A -85,B 0,C 180,E1 -308.235,E2 -308.235} C_VEL
LIN {X 0,Y 608.418,Z 713.095,A -85,B 0,C 180,E1 -309.444,E2 -309.444} C_VEL
LIN {X 0,Y 608.434,Z 710.687,A -85,B 0,C 180,E1 -310.74,E2 -310.74} C_VEL
LIN {X 0,Y 608.45,Z 707.941,A -85,B 0,C 180,E1 -311.673,E2 -311.673} C_VEL
LIN {X 0,Y 608.442,Z 704.219,A -85,B 0,C 180,E1 -312.619,E2 -312.619} C_VEL
LIN {X 0,Y 608.453,Z 699.508,A -85,B 0,C 180,E1 -313.561,E2 -313.561} C_VEL
LIN {X 0,Y 608.459,Z 692.684,A -85,B 0,C 180,E1 -314.648,E2 -314.648} C_VEL
LIN {X 0,Y 608.469,Z 683.971,A -85,B 0,C 180,E1 -315.735,E2 -315.735} C_VEL
LIN {X 0,Y 608.476,Z 675.475,A -85,B 0,C 180,E1 -316.595,E2 -316.595} C_VEL
LIN {X 0,Y 608.481,Z 665.945,A -85,B 0,C 180,E1 -317.384,E2 -317.384} C_VEL
LIN {X 0,Y 608.493,Z 654.651,A -85,B 0,C 180,E1 -318.136,E2 -318.136} C_VEL
LIN {X 0,Y 608.513,Z 642.518,A -85,B 0,C 180,E1 -318.773,E2 -318.773} C_VEL
LIN {X 0,Y 608.536,Z 629.913,A -85,B 0,C 180,E1 -319.269,E2 -319.269} C_VEL
LIN {X 0,Y 608.488,Z 624.693,A -85,B 0,C 180,E1 -319.444,E2 -319.444} C_VEL
LIN {X 0,Y 608.472,Z 624.685,A -85,B 0,C 180,E1 -322.254,E2 -322.254} C_VEL
LIN {X 0,Y 608.451,Z 624.69,A -85,B 0,C 180,E1 -325.094,E2 -325.094} C_VEL
LIN {X 0,Y 608.47,Z 624.691,A -85,B 0,C 180,E1 -327.906,E2 -327.906} C_VEL
LIN {X 0,Y 608.469,Z 624.687,A -85,B 0,C 180,E1 -330.221,E2 -330.221} C_VEL
LIN {X 0,Y 608.476,Z 624.684,A -85,B 0,C 180,E1 -332.793,E2 -332.793} C_VEL
LIN {X 0,Y 608.456,Z 624.692,A -85,B 0,C 180,E1 -335.429,E2 -335.429} C_VEL
LIN {X 0,Y 608.463,Z 624.688,A -85,B 0,C 180,E1 -338.308,E2 -338.308} C_VEL
LIN {X 0,Y 608.454,Z 624.688,A -85,B 0,C 180,E1 -341.13,E2 -341.13} C_VEL
LIN {X 0,Y 608.465,Z 624.696,A -85,B 0,C 180,E1 -343.906,E2 -343.906} C_VEL
LIN {X 0,Y 608.457,Z 624.687,A -85,B 0,C 180,E1 -346.644,E2 -346.644} C_VEL
LIN {X 0,Y 608.467,Z 624.687,A -85,B 0,C 180,E1 -349.35,E2 -349.35} C_VEL
LIN {X 0,Y 608.484,Z 624.693,A -85,B 0,C 180,E1 -352.033,E2 -352.033} C_VEL
LIN {X 0,Y 608.458,Z 624.687,A -85,B 0,C 180,E1 -354.698,E2 -354.698} C_VEL
LIN {X 0,Y 608.483,Z 624.684,A -85,B 0,C 180,E1 -357.352,E2 -357.352} C_VEL
LIN {X 0,Y 608.48,Z 624.693,A -85,B 0,C 180,E1 -360,E2 -360} C_VEL
LIN {X 0,Y 608.484,Z 624.685,A -85,B 0,C 180,E1 -362.648,E2 -362.648} C_VEL
LIN {X 0,Y 608.458,Z 624.686,A -85,B 0,C 180,E1 -365.302,E2 -365.302} C_VEL
LIN {X 0,Y 608.484,Z 624.69,A -85,B 0,C 180,E1 -367.967,E2 -367.967} C_VEL
LIN {X 0,Y 608.468,Z 624.686,A -85,B 0,C 180,E1 -370.956,E2 -370.956} C_VEL
LIN {X 0,Y 608.459,Z 624.686,A -85,B 0,C 180,E1 -373.357,E2 -373.357} C_VEL
LIN {X 0,Y 608.465,Z 624.693,A -85,B 0,C 180,E1 -376.094,E2 -376.094} C_VEL
LIN {X 0,Y 608.453,Z 624.689,A -85,B 0,C 180,E1 -378.87,E2 -378.87} C_VEL
LIN {X 0,Y 608.466,Z 624.686,A -85,B 0,C 180,E1 -381.692,E2 -381.692} C_VEL
LIN {X 0,Y 608.459,Z 624.694,A -85,B 0,C 180,E1 -384.571,E2 -384.571} C_VEL
LIN {X 0,Y 608.476,Z 624.684,A -85,B 0,C 180,E1 -387.207,E2 -387.207} C_VEL
LIN {X 0,Y 608.469,Z 624.687,A -85,B 0,C 180,E1 -389.972,E2 -389.972} C_VEL
LIN {X 0,Y 608.458,Z 624.691,A -85,B 0,C 180,E1 -392.88,E2 -392.88} C_VEL
LIN {X 0,Y 608.436,Z 624.69,A -85,B 0,C 180,E1 -395.278,E2 -395.278} C_VEL
LIN {X 0,Y 608.472,Z 624.685,A -85,B 0,C 180,E1 -397.746,E2 -397.746} C_VEL
LIN {X 0,Y 608.457,Z 624.692,A -85,B 0,C 180,E1 -400.33,E2 -400.33} C_VEL
LIN {X 0,Y 608.484,Z 624.684,A -85,B 0,C 180,E1 -403.31,E2 -403.31} C_VEL
LIN {X 0,Y 608.469,Z 624.687,A -85,B 0,C 180,E1 -406.13,E2 -406.13} C_VEL
LIN {X 0,Y 608.455,Z 624.697,A -85,B 0,C 180,E1 -408.823,E2 -408.823} C_VEL
LIN {X 0,Y 608.436,Z 624.691,A -85,B 0,C 180,E1 -411.409,E2 -411.409} C_VEL
LIN {X 0,Y 608.461,Z 624.687,A -85,B 0,C 180,E1 -414.014,E2 -414.014} C_VEL
LIN {X 0,Y 608.468,Z 624.735,A -85,B 0,C 180,E1 -414.149,E2 -414.149} C_VEL
LIN {X 0,Y 608.672,Z 631.758,A -85,B 0,C 180,E1 -415.544,E2 -415.544} C_VEL
LIN {X 0,Y 608.642,Z 645.452,A -85,B 0,C 180,E1 -418.305,E2 -418.305} C_VEL
LIN {X 0,Y 608.596,Z 659.147,A -85,B 0,C 180,E1 -420.987,E2 -420.987} C_VEL
LIN {X 0,Y 608.558,Z 672.842,A -85,B 0,C 180,E1 -423.601,E2 -423.601} C_VEL
LIN {X 0,Y 608.532,Z 686.537,A -85,B 0,C 180,E1 -426.158,E2 -426.158} C_VEL
LIN {X 0,Y 608.531,Z 700.232,A -85,B 0,C 180,E1 -428.666,E2 -428.666} C_VEL
LIN {X 0,Y 608.493,Z 716.299,A -85,B 0,C 180,E1 -431.555,E2 -431.555} C_VEL
LIN {X 0,Y 608.478,Z 731.534,A -85,B 0,C 180,E1 -434.251,E2 -434.251} C_VEL
LIN {X 0,Y 608.462,Z 747.185,A -85,B 0,C 180,E1 -436.983,E2 -436.983} C_VEL
LIN {X 0,Y 608.44,Z 754.155,A -85,B 0,C 180,E1 -438.19,E2 -438.19} C_VEL
LIN {X 0,Y 608.536,Z 768.255,A -85,B 0,C 180,E1 -438.445,E2 -438.445} C_VEL
LIN {X 0,Y 608.531,Z 780.954,A -85,B 0,C 180,E1 -438.81,E2 -438.81} C_VEL
LIN {X 0,Y 608.498,Z 792.679,A -85,B 0,C 180,E1 -439.279,E2 -439.279} C_VEL
LIN {X 0,Y 608.486,Z 803.751,A -85,B 0,C 180,E1 -439.855,E2 -439.855} C_VEL
LIN {X 0,Y 608.504,Z 815.248,A -85,B 0,C 180,E1 -440.611,E2 -440.611} C_VEL
LIN {X 0,Y 608.472,Z 824.533,A -85,B 0,C 180,E1 -441.364,E2 -441.364} C_VEL
LIN {X 0,Y 608.456,Z 832.986,A -85,B 0,C 180,E1 -442.2,E2 -442.2} C_VEL
LIN {X 0,Y 608.462,Z 841.233,A -85,B 0,C 180,E1 -443.2,E2 -443.2} C_VEL
LIN {X 0,Y 608.437,Z 847.875,A -85,B 0,C 180,E1 -444.199,E2 -444.199} C_VEL
LIN {X 0,Y 608.432,Z 853.949,A -85,B 0,C 180,E1 -445.362,E2 -445.362} C_VEL
LIN {X 0,Y 608.449,Z 857.895,A -85,B 0,C 180,E1 -446.357,E2 -446.357} C_VEL
LIN {X 0,Y 608.425,Z 860.808,A -85,B 0,C 180,E1 -447.351,E2 -447.351} C_VEL
LIN {X 0,Y 608.441,Z 862.201,A -85,B 0,C 180,E1 -448.014,E2 -448.014} C_VEL
LIN {X 0,Y 608.439,Z 863.783,A -85,B 0,C 180,E1 -449.338,E2 -449.338} C_VEL
LIN {X 0,Y 608.434,Z 864,A -85,B 0,C 180,E1 -450,E2 -450} C_VEL
LIN {X 0,Y 608.448,Z 863.184,A -85,B 0,C 180,E1 -451.323,E2 -451.323} C_VEL
LIN {X 0,Y 608.441,Z 862.202,A -85,B 0,C 180,E1 -451.985,E2 -451.985} C_VEL
LIN {X 0,Y 608.425,Z 860.81,A -85,B 0,C 180,E1 -452.648,E2 -452.648} C_VEL
LIN {X 0,Y 608.449,Z 857.897,A -85,B 0,C 180,E1 -453.642,E2 -453.642} C_VEL
LIN {X 0,Y 608.432,Z 853.952,A -85,B 0,C 180,E1 -454.637,E2 -454.637} C_VEL
LIN {X 0,Y 608.437,Z 847.879,A -85,B 0,C 180,E1 -455.8,E2 -455.8} C_VEL
LIN {X 0,Y 608.462,Z 841.238,A -85,B 0,C 180,E1 -456.799,E2 -456.799} C_VEL
LIN {X 0,Y 608.455,Z 832.993,A -85,B 0,C 180,E1 -457.8,E2 -457.8} C_VEL
LIN {X 0,Y 608.472,Z 824.541,A -85,B 0,C 180,E1 -458.635,E2 -458.635} C_VEL
LIN {X 0,Y 608.48,Z 814.096,A -85,B 0,C 180,E1 -459.473,E2 -459.473} C_VEL
LIN {X 0,Y 608.485,Z 803.763,A -85,B 0,C 180,E1 -460.144,E2 -460.144} C_VEL
LIN {X 0,Y 608.5,Z 792.297,A -85,B 0,C 180,E1 -460.739,E2 -460.739} C_VEL
LIN {X 0,Y 608.536,Z 779.952,A -85,B 0,C 180,E1 -461.223,E2 -461.223} C_VEL
LIN {X 0,Y 608.534,Z 766.459,A -85,B 0,C 180,E1 -461.597,E2 -461.597} C_VEL
LIN {X 0,Y 608.439,Z 754.159,A -85,B 0,C 180,E1 -461.81,E2 -461.81} C_VEL
LIN {X 0,Y 608.467,Z 739.364,A -85,B 0,C 180,E1 -464.378,E2 -464.378} C_VEL
LIN {X 0,Y 608.479,Z 723.713,A -85,B 0,C 180,E1 -467.129,E2 -467.129} C_VEL
LIN {X 0,Y 608.508,Z 708.061,A -85,B 0,C 180,E1 -469.92,E2 -469.92} C_VEL
LIN {X 0,Y 608.528,Z 693.882,A -85,B 0,C 180,E1 -472.491,E2 -472.491} C_VEL
LIN {X 0,Y 608.563,Z 678.715,A -85,B 0,C 180,E1 -475.295,E2 -475.295} C_VEL
LIN {X 0,Y 608.583,Z 665.021,A -85,B 0,C 180,E1 -477.884,E2 -477.884} C_VEL
LIN {X 0,Y 608.619,Z 651.326,A -85,B 0,C 180,E1 -480.536,E2 -480.536} C_VEL
LIN {X 0,Y 608.659,Z 639.587,A -85,B 0,C 180,E1 -482.867,E2 -482.867} C_VEL
LIN {X 0,Y 608.646,Z 626.773,A -85,B 0,C 180,E1 -485.455,E2 -485.455} C_VEL
LIN {X 0,Y 608.459,Z 624.69,A -85,B 0,C 180,E1 -485.886,E2 -485.886} C_VEL
LIN {X 0,Y 608.473,Z 624.69,A -85,B 0,C 180,E1 -488.587,E2 -488.587} C_VEL
LIN {X 0,Y 608.461,Z 624.69,A -85,B 0,C 180,E1 -491.342,E2 -491.342} C_VEL
LIN {X 0,Y 608.45,Z 624.692,A -85,B 0,C 180,E1 -494.263,E2 -494.263} C_VEL
LIN {X 0,Y 608.452,Z 624.691,A -85,B 0,C 180,E1 -497.04,E2 -497.04} C_VEL
LIN {X 0,Y 608.453,Z 624.689,A -85,B 0,C 180,E1 -499.696,E2 -499.696} C_VEL
LIN {X 0,Y 608.475,Z 624.695,A -85,B 0,C 180,E1 -502.254,E2 -502.254} C_VEL
LIN {X 0,Y 608.434,Z 624.692,A -85,B 0,C 180,E1 -504.722,E2 -504.722} C_VEL
LIN {X 0,Y 608.453,Z 624.691,A -85,B 0,C 180,E1 -507.478,E2 -507.478} C_VEL
LIN {X 0,Y 608.469,Z 624.69,A -85,B 0,C 180,E1 -510.22,E2 -510.22} C_VEL
LIN {X 0,Y 608.475,Z 624.685,A -85,B 0,C 180,E1 -512.792,E2 -512.792} C_VEL
LIN {X 0,Y 608.458,Z 624.695,A -85,B 0,C 180,E1 -515.429,E2 -515.429} C_VEL
LIN {X 0,Y 608.463,Z 624.687,A -85,B 0,C 180,E1 -518.308,E2 -518.308} C_VEL
LIN {X 0,Y 608.452,Z 624.696,A -85,B 0,C 180,E1 -521.13,E2 -521.13} C_VEL
LIN {X 0,Y 608.456,Z 624.688,A -85,B 0,C 180,E1 -523.906,E2 -523.906} C_VEL
LIN {X 0,Y 608.467,Z 624.691,A -85,B 0,C 180,E1 -526.644,E2 -526.644} C_VEL
LIN {X 0,Y 608.465,Z 624.689,A -85,B 0,C 180,E1 -529.35,E2 -529.35} C_VEL
LIN {X 0,Y 608.475,Z 624.687,A -85,B 0,C 180,E1 -532.033,E2 -532.033} C_VEL
LIN {X 0,Y 608.458,Z 624.695,A -85,B 0,C 180,E1 -534.698,E2 -534.698} C_VEL
LIN {X 0,Y 608.483,Z 624.684,A -85,B 0,C 180,E1 -537.352,E2 -537.352} C_VEL
LIN {X 0,Y 608.472,Z 624.691,A -85,B 0,C 180,E1 -540,E2 -540} C_VEL
LIN {X 0,Y 608.483,Z 624.687,A -85,B 0,C 180,E1 -542.648,E2 -542.648} C_VEL
LIN {X 0,Y 608.492,Z 624.804,A -85,B 0,C 180,E1 -545.468,E2 -545.468} C_VEL
LIN {X 0,Y 608.584,Z 630.135,A -85,B 0,C 180,E1 -546.723,E2 -546.723} C_VEL
LIN {X 0,Y 608.556,Z 639.946,A -85,B 0,C 180,E1 -549.245,E2 -549.245} C_VEL
LIN {X 0,Y 607.918,Z 642.12,A -85,B 0,C 180,E1 -549.758,E2 -549.758} C_VEL
LIN {X 0,Y 602.266,Z 649.914,A -85,B 0,C 180,E1 -551.404,E2 -551.404} C_VEL
LIN {X 0,Y 601.589,Z 652.137,A -85,B 0,C 180,E1 -551.924,E2 -551.924} C_VEL
LIN {X 0,Y 601.527,Z 664.216,A -85,B 0,C 180,E1 -554.894,E2 -554.894} C_VEL
LIN {X 0,Y 601.502,Z 675.839,A -85,B 0,C 180,E1 -557.685,E2 -557.685} C_VEL
LIN {X 0,Y 601.463,Z 686.372,A -85,B 0,C 180,E1 -560.164,E2 -560.164} C_VEL
LIN {X 0,Y 601.426,Z 698.836,A -85,B 0,C 180,E1 -563.046,E2 -563.046} C_VEL
LIN {X 0,Y 601.401,Z 711.232,A -85,B 0,C 180,E1 -565.867,E2 -565.867} C_VEL
LIN {X 0,Y 601.382,Z 723.533,A -85,B 0,C 180,E1 -568.629,E2 -568.629} C_VEL
LIN {X 0,Y 601.372,Z 725.721,A -85,B 0,C 180,E1 -569.117,E2 -569.117} C_VEL
LIN {X 0,Y 601.586,Z 735.543,A -85,B 0,C 180,E1 -569.291,E2 -569.291} C_VEL
LIN {X 0,Y 601.556,Z 748.005,A -85,B 0,C 180,E1 -569.626,E2 -569.626} C_VEL
LIN {X 0,Y 601.518,Z 760.287,A -85,B 0,C 180,E1 -570.092,E2 -570.092} C_VEL
LIN {X 0,Y 601.51,Z 770.855,A -85,B 0,C 180,E1 -570.615,E2 -570.615} C_VEL
LIN {X 0,Y 601.457,Z 781.541,A -85,B 0,C 180,E1 -571.276,E2 -571.276} C_VEL
LIN {X 0,Y 601.433,Z 791.259,A -85,B 0,C 180,E1 -572.021,E2 -572.021} C_VEL
LIN {X 0,Y 601.409,Z 801.451,A -85,B 0,C 180,E1 -572.987,E2 -572.987} C_VEL
LIN {X 0,Y 601.402,Z 809.519,A -85,B 0,C 180,E1 -573.933,E2 -573.933} C_VEL
LIN {X 0,Y 601.37,Z 816.432,A -85,B 0,C 180,E1 -574.935,E2 -574.935} C_VEL
LIN {X 0,Y 601.379,Z 822.307,A -85,B 0,C 180,E1 -576.004,E2 -576.004} C_VEL
LIN {X 0,Y 601.344,Z 826.505,A -85,B 0,C 180,E1 -576.977,E2 -576.977} C_VEL
LIN {X 0,Y 601.338,Z 830.57,A -85,B 0,C 180,E1 -578.274,E2 -578.274} C_VEL
LIN {X 0,Y 601.316,Z 832.97,A -85,B 0,C 180,E1 -579.522,E2 -579.522} C_VEL
LIN {X 0,Y 601.314,Z 833.969,A -85,B 0,C 180,E1 -580.883,E2 -580.883} C_VEL
LIN {X 0,Y 601.322,Z 833.742,A -85,B 0,C 180,E1 -581.774,E2 -581.774} C_VEL
LIN {X 0,Y 601.34,Z 832.821,A -85,B 0,C 180,E1 -582.677,E2 -582.677} C_VEL
LIN {X 0,Y 601.341,Z 831.102,A -85,B 0,C 180,E1 -583.594,E2 -583.594} C_VEL
LIN {X 0,Y 601.33,Z 828.541,A -85,B 0,C 180,E1 -584.527,E2 -584.527} C_VEL
LIN {X 0,Y 601.369,Z 824.059,A -85,B 0,C 180,E1 -585.712,E2 -585.712} C_VEL
LIN {X 0,Y 601.372,Z 818.065,A -85,B 0,C 180,E1 -586.883,E2 -586.883} C_VEL
LIN {X 0,Y 601.369,Z 810.485,A -85,B 0,C 180,E1 -588.027,E2 -588.027} C_VEL
LIN {X 0,Y 601.383,Z 802.914,A -85,B 0,C 180,E1 -588.946,E2 -588.946} C_VEL
LIN {X 0,Y 601.433,Z 794.388,A -85,B 0,C 180,E1 -589.796,E2 -589.796} C_VEL
LIN {X 0,Y 601.447,Z 783.551,A -85,B 0,C 180,E1 -590.67,E2 -590.67} C_VEL
LIN {X 0,Y 601.486,Z 772.1,A -85,B 0,C 180,E1 -591.407,E2 -591.407} C_VEL
LIN {X 0,Y 601.5,Z 760.143,A -85,B 0,C 180,E1 -592.005,E2 -592.005} C_VEL
LIN {X 0,Y 601.563,Z 747.342,A -85,B 0,C 180,E1 -592.486,E2 -592.486} C_VEL
LIN {X 0,Y 601.601,Z 734.496,A -85,B 0,C 180,E1 -592.821,E2 -592.821} C_VEL
LIN {X 0,Y 601.362,Z 725.742,A -85,B 0,C 180,E1 -592.973,E2 -592.973} C_VEL
LIN {X 0,Y 601.407,Z 714.545,A -85,B 0,C 180,E1 -595.476,E2 -595.476} C_VEL
LIN {X 0,Y 601.423,Z 702.198,A -85,B 0,C 180,E1 -598.275,E2 -598.275} C_VEL
LIN {X 0,Y 601.465,Z 690.589,A -85,B 0,C 180,E1 -600.945,E2 -600.945} C_VEL
LIN {X 0,Y 601.491,Z 677.897,A -85,B 0,C 180,E1 -603.917,E2 -603.917} C_VEL
LIN {X 0,Y 601.533,Z 666.693,A -85,B 0,C 180,E1 -606.595,E2 -606.595} C_VEL
LIN {X 0,Y 601.561,Z 656.156,A -85,B 0,C 180,E1 -609.169,E2 -609.169} C_VEL
LIN {X 0,Y 601.591,Z 646.377,A -85,B 0,C 180,E1 -611.614,E2 -611.614} C_VEL
LIN {X 0,Y 601.66,Z 635.463,A -85,B 0,C 180,E1 -614.416,E2 -614.416} C_VEL
LIN {X 0,Y 601.53,Z 626.172,A -85,B 0,C 180,E1 -616.659,E2 -616.659} C_VEL
LIN {X 0,Y 601.468,Z 625.565,A -85,B 0,C 180,E1 -616.83,E2 -616.83} C_VEL
LIN {X 0,Y 601.413,Z 625.571,A -85,B 0,C 180,E1 -619.224,E2 -619.224} C_VEL
LIN {X 0,Y 601.441,Z 625.567,A -85,B 0,C 180,E1 -621.94,E2 -621.94} C_VEL
LIN {X 0,Y 601.43,Z 625.569,A -85,B 0,C 180,E1 -624.636,E2 -624.636} C_VEL
LIN {X 0,Y 601.436,Z 625.568,A -85,B 0,C 180,E1 -627.321,E2 -627.321} C_VEL
LIN {X 0,Y 601.45,Z 625.566,A -85,B 0,C 180,E1 -630,E2 -630} C_VEL
LIN {X 0,Y 601.436,Z 625.568,A -85,B 0,C 180,E1 -632.679,E2 -632.679} C_VEL
LIN {X 0,Y 601.428,Z 625.569,A -85,B 0,C 180,E1 -635.364,E2 -635.364} C_VEL
LIN {X 0,Y 601.444,Z 625.566,A -85,B 0,C 180,E1 -638.061,E2 -638.061} C_VEL
LIN {X 0,Y 601.424,Z 625.57,A -85,B 0,C 180,E1 -641.011,E2 -641.011} C_VEL
LIN {X 0,Y 601.425,Z 625.569,A -85,B 0,C 180,E1 -643.516,E2 -643.516} C_VEL
LIN {X 0,Y 601.443,Z 625.567,A -85,B 0,C 180,E1 -646.287,E2 -646.287} C_VEL
LIN {X 0,Y 601.417,Z 625.572,A -85,B 0,C 180,E1 -649.099,E2 -649.099} C_VEL
LIN {X 0,Y 601.41,Z 625.571,A -85,B 0,C 180,E1 -651.239,E2 -651.239} C_VEL
LIN {X 0,Y 601.453,Z 625.566,A -85,B 0,C 180,E1 -654.141,E2 -654.141} C_VEL
LIN {X 0,Y 601.435,Z 625.66,A -85,B 0,C 180,E1 -656.549,E2 -656.549} C_VEL
LIN {X 0,Y 601.517,Z 638.48,A -85,B 0,C 180,E1 -657.014,E2 -657.014} C_VEL
LIN {X 0,Y 601.504,Z 651.203,A -85,B 0,C 180,E1 -657.634,E2 -657.634} C_VEL
LIN {X 0,Y 601.477,Z 662.427,A -85,B 0,C 180,E1 -658.339,E2 -658.339} C_VEL
LIN {X 0,Y 601.438,Z 671.689,A -85,B 0,C 180,E1 -659.059,E2 -659.059} C_VEL
LIN {X 0,Y 601.405,Z 681.192,A -85,B 0,C 180,E1 -659.961,E2 -659.961} C_VEL
LIN {X 0,Y 601.383,Z 689.602,A -85,B 0,C 180,E1 -660.944,E2 -660.944} C_VEL
LIN {X 0,Y 601.368,Z 696.382,A -85,B 0,C 180,E1 -661.926,E2 -661.926} C_VEL
LIN {X 0,Y 601.346,Z 702.219,A -85,B 0,C 180,E1 -662.985,E2 -662.985} C_VEL
LIN {X 0,Y 601.342,Z 707.048,A -85,B 0,C 180,E1 -664.124,E2 -664.124} C_VEL
LIN {X 0,Y 601.323,Z 710.118,A -85,B 0,C 180,E1 -665.102,E2 -665.102} C_VEL
LIN {X 0,Y 601.316,Z 712.553,A -85,B 0,C 180,E1 -666.249,E2 -666.249} C_VEL
LIN {X 0,Y 601.33,Z 713.82,A -85,B 0,C 180,E1 -667.427,E2 -667.427} C_VEL
LIN {X 0,Y 601.315,Z 713.911,A -85,B 0,C 180,E1 -668.457,E2 -668.457} C_VEL
LIN {X 0,Y 601.313,Z 713.025,A -85,B 0,C 180,E1 -669.521,E2 -669.521} C_VEL
LIN {X 0,Y 601.33,Z 710.399,A -85,B 0,C 180,E1 -670.881,E2 -670.881} C_VEL
LIN {X 0,Y 601.359,Z 706.274,A -85,B 0,C 180,E1 -672.176,E2 -672.176} C_VEL
LIN {X 0,Y 601.344,Z 701.029,A -85,B 0,C 180,E1 -673.343,E2 -673.343} C_VEL
LIN {X 0,Y 601.375,Z 695.594,A -85,B 0,C 180,E1 -674.289,E2 -674.289} C_VEL
LIN {X 0,Y 601.383,Z 688.049,A -85,B 0,C 180,E1 -675.341,E2 -675.341} C_VEL
LIN {X 0,Y 601.415,Z 679.574,A -85,B 0,C 180,E1 -676.297,E2 -676.297} C_VEL
LIN {X 0,Y 601.431,Z 669.457,A -85,B 0,C 180,E1 -677.217,E2 -677.217} C_VEL
LIN {X 0,Y 601.486,Z 658.505,A -85,B 0,C 180,E1 -678.015,E2 -678.015} C_VEL
LIN {X 0,Y 601.505,Z 648.213,A -85,B 0,C 180,E1 -678.618,E2 -678.618} C_VEL
LIN {X 0,Y 601.54,Z 635.96,A -85,B 0,C 180,E1 -679.18,E2 -679.18} C_VEL
LIN {X 0,Y 601.44,Z 625.571,A -85,B 0,C 180,E1 -679.563,E2 -679.563} C_VEL
LIN {X 0,Y 601.427,Z 625.57,A -85,B 0,C 180,E1 -681.733,E2 -681.733} C_VEL
LIN {X 0,Y 601.387,Z 625.568,A -85,B 0,C 180,E1 -684.245,E2 -684.245} C_VEL
LIN {X 0,Y 601.42,Z 625.563,A -85,B 0,C 180,E1 -686.686,E2 -686.686} C_VEL
LIN {X 0,Y 601.416,Z 625.566,A -85,B 0,C 180,E1 -689.058,E2 -689.058} C_VEL
LIN {X 0,Y 601.437,Z 625.566,A -85,B 0,C 180,E1 -691.373,E2 -691.373} C_VEL
LIN {X 0,Y 601.411,Z 625.568,A -85,B 0,C 180,E1 -694.133,E2 -694.133} C_VEL
LIN {X 0,Y 601.418,Z 625.563,A -85,B 0,C 180,E1 -696.59,E2 -696.59} C_VEL
LIN {X 0,Y 601.436,Z 625.567,A -85,B 0,C 180,E1 -699.478,E2 -699.478} C_VEL
LIN {X 0,Y 601.395,Z 625.569,A -85,B 0,C 180,E1 -702.312,E2 -702.312} C_VEL
LIN {X 0,Y 601.412,Z 625.566,A -85,B 0,C 180,E1 -704.409,E2 -704.409} C_VEL
LIN {X 0,Y 601.421,Z 625.564,A -85,B 0,C 180,E1 -707.172,E2 -707.172} C_VEL
LIN {X 0,Y 601.434,Z 625.572,A -85,B 0,C 180,E1 -709.905,E2 -709.905} C_VEL
LIN {X 0,Y 601.439,Z 625.562,A -85,B 0,C 180,E1 -712.615,E2 -712.615} C_VEL
LIN {X 0,Y 601.431,Z 625.563,A -85,B 0,C 180,E1 -715.308,E2 -715.308} C_VEL
LIN {X 0,Y 601.438,Z 625.571,A -85,B 0,C 180,E1 -717.991,E2 -717.991} C_VEL
LIN {X 0,Y 601.451,Z 625.561,A -85,B 0,C 180,E1 -720.67,E2 -720.67} C_VEL
LIN {X 0,Y 601.427,Z 625.563,A -85,B 0,C 180,E1 -723.35,E2 -723.35} C_VEL
LIN {X 0,Y 601.416,Z 625.572,A -85,B 0,C 180,E1 -726.037,E2 -726.037} C_VEL
LIN {X 0,Y 601.439,Z 625.563,A -85,B 0,C 180,E1 -728.738,E2 -728.738} C_VEL
LIN {X 0,Y 601.434,Z 625.562,A -85,B 0,C 180,E1 -731.458,E2 -731.458} C_VEL
LIN {X 0,Y 601.421,Z 625.573,A -85,B 0,C 180,E1 -734.206,E2 -734.206} C_VEL
LIN {X 0,Y 601.432,Z 625.562,A -85,B 0,C 180,E1 -736.986,E2 -736.986} C_VEL
LIN {X 0,Y 601.406,Z 625.567,A -85,B 0,C 180,E1 -739.81,E2 -739.81} C_VEL
LIN {X 0,Y 601.413,Z 625.569,A -85,B 0,C 180,E1 -742.683,E2 -742.683} C_VEL
LIN {X 0,Y 601.405,Z 625.568,A -85,B 0,C 180,E1 -744.879,E2 -744.879} C_VEL
LIN {X 0,Y 601.415,Z 625.564,A -85,B 0,C 180,E1 -747.362,E2 -747.362} C_VEL
LIN {X 0,Y 601.43,Z 625.567,A -85,B 0,C 180,E1 -750.164,E2 -750.164} C_VEL
LIN {X 0,Y 601.426,Z 625.57,A -85,B 0,C 180,E1 -752.716,E2 -752.716} C_VEL
LIN {X 0,Y 601.392,Z 625.569,A -85,B 0,C 180,E1 -755.112,E2 -755.112} C_VEL
LIN {X 0,Y 601.438,Z 625.561,A -85,B 0,C 180,E1 -757.419,E2 -757.419} C_VEL
LIN {X 0,Y 601.414,Z 625.565,A -85,B 0,C 180,E1 -759.995,E2 -759.995} C_VEL
LIN {X 0,Y 601.416,Z 625.575,A -85,B 0,C 180,E1 -762.67,E2 -762.67} C_VEL
LIN {X 0,Y 601.399,Z 625.566,A -85,B 0,C 180,E1 -765.468,E2 -765.468} C_VEL
LIN {X 0,Y 601.425,Z 625.568,A -85,B 0,C 180,E1 -768.407,E2 -768.407} C_VEL
LIN {X 0,Y 601.429,Z 625.573,A -85,B 0,C 180,E1 -770.875,E2 -770.875} C_VEL
LIN {X 0,Y 601.402,Z 625.57,A -85,B 0,C 180,E1 -773.417,E2 -773.417} C_VEL
LIN {X 0,Y 601.451,Z 625.71,A -85,B 0,C 180,E1 -773.98,E2 -773.98} C_VEL
LIN {X 0,Y 601.786,Z 631.438,A -85,B 0,C 180,E1 -775.093,E2 -775.093} C_VEL
LIN {X 0,Y 601.792,Z 641.111,A -85,B 0,C 180,E1 -777.021,E2 -777.021} C_VEL
LIN {X 0,Y 601.759,Z 653.28,A -85,B 0,C 180,E1 -779.467,E2 -779.467} C_VEL
LIN {X 0,Y 601.679,Z 666.973,A -85,B 0,C 180,E1 -782.145,E2 -782.145} C_VEL
LIN {X 0,Y 601.605,Z 680.668,A -85,B 0,C 180,E1 -784.761,E2 -784.761} C_VEL
LIN {X 0,Y 601.569,Z 694.564,A -85,B 0,C 180,E1 -787.36,E2 -787.36} C_VEL
LIN {X 0,Y 601.512,Z 710.014,A -85,B 0,C 180,E1 -790.194,E2 -790.194} C_VEL
LIN {X 0,Y 601.445,Z 725.665,A -85,B 0,C 180,E1 -793.014,E2 -793.014} C_VEL
LIN {X 0,Y 601.434,Z 739.36,A -85,B 0,C 180,E1 -795.449,E2 -795.449} C_VEL
LIN {X 0,Y 601.408,Z 754.155,A -85,B 0,C 180,E1 -798.05,E2 -798.05} C_VEL
LIN {X 0,Y 601.595,Z 767.341,A -85,B 0,C 180,E1 -798.288,E2 -798.288} C_VEL
LIN {X 0,Y 601.566,Z 780.432,A -85,B 0,C 180,E1 -798.662,E2 -798.662} C_VEL
LIN {X 0,Y 601.512,Z 792.678,A -85,B 0,C 180,E1 -799.153,E2 -799.153} C_VEL
LIN {X 0,Y 601.489,Z 803.752,A -85,B 0,C 180,E1 -799.736,E2 -799.736} C_VEL
LIN {X 0,Y 601.462,Z 815.249,A -85,B 0,C 180,E1 -800.5,E2 -800.5} C_VEL
LIN {X 0,Y 601.436,Z 824.533,A -85,B 0,C 180,E1 -801.262,E2 -801.262} C_VEL
LIN {X 0,Y 601.4,Z 832.987,A -85,B 0,C 180,E1 -802.107,E2 -802.107} C_VEL
LIN {X 0,Y 601.382,Z 841.233,A -85,B 0,C 180,E1 -803.12,E2 -803.12} C_VEL
LIN {X 0,Y 601.372,Z 847.875,A -85,B 0,C 180,E1 -804.13,E2 -804.13} C_VEL
LIN {X 0,Y 601.336,Z 853.948,A -85,B 0,C 180,E1 -805.307,E2 -805.307} C_VEL
LIN {X 0,Y 601.368,Z 857.895,A -85,B 0,C 180,E1 -806.314,E2 -806.314} C_VEL
LIN {X 0,Y 601.325,Z 860.808,A -85,B 0,C 180,E1 -807.32,E2 -807.32} C_VEL
LIN {X 0,Y 601.34,Z 862.201,A -85,B 0,C 180,E1 -807.99,E2 -807.99} C_VEL
LIN {X 0,Y 601.339,Z 863.783,A -85,B 0,C 180,E1 -809.33,E2 -809.33} C_VEL
LIN {X 0,Y 601.335,Z 864,A -85,B 0,C 180,E1 -810,E2 -810} C_VEL
LIN {X 0,Y 601.348,Z 863.184,A -85,B 0,C 180,E1 -811.339,E2 -811.339} C_VEL
LIN {X 0,Y 601.34,Z 862.202,A -85,B 0,C 180,E1 -812.009,E2 -812.009} C_VEL
LIN {X 0,Y 601.325,Z 860.81,A -85,B 0,C 180,E1 -812.679,E2 -812.679} C_VEL
LIN {X 0,Y 601.368,Z 857.897,A -85,B 0,C 180,E1 -813.685,E2 -813.685} C_VEL
LIN {X 0,Y 601.336,Z 853.952,A -85,B 0,C 180,E1 -814.692,E2 -814.692} C_VEL
LIN {X 0,Y 601.372,Z 847.879,A -85,B 0,C 180,E1 -815.869,E2 -815.869} C_VEL
LIN {X 0,Y 601.381,Z 841.238,A -85,B 0,C 180,E1 -816.879,E2 -816.879} C_VEL
LIN {X 0,Y 601.4,Z 832.993,A -85,B 0,C 180,E1 -817.892,E2 -817.892} C_VEL
LIN {X 0,Y 601.436,Z 824.541,A -85,B 0,C 180,E1 -818.737,E2 -818.737} C_VEL
LIN {X 0,Y 601.446,Z 814.098,A -85,B 0,C 180,E1 -819.585,E2 -819.585} C_VEL
LIN {X 0,Y 601.488,Z 803.764,A -85,B 0,C 180,E1 -820.264,E2 -820.264} C_VEL
LIN {X 0,Y 601.532,Z 791.922,A -85,B 0,C 180,E1 -820.882,E2 -820.882} C_VEL
LIN {X 0,Y 601.562,Z 779.29,A -85,B 0,C 180,E1 -821.376,E2 -821.376} C_VEL
LIN {X 0,Y 601.585,Z 766.459,A -85,B 0,C 180,E1 -821.732,E2 -821.732} C_VEL
LIN {X 0,Y 601.408,Z 754.159,A -85,B 0,C 180,E1 -821.95,E2 -821.95} C_VEL
LIN {X 0,Y 601.434,Z 737.407,A -85,B 0,C 180,E1 -824.896,E2 -824.896} C_VEL
LIN {X 0,Y 601.488,Z 721.756,A -85,B 0,C 180,E1 -827.685,E2 -827.685} C_VEL
LIN {X 0,Y 601.505,Z 706.105,A -85,B 0,C 180,E1 -830.519,E2 -830.519} C_VEL
LIN {X 0,Y 601.568,Z 690.454,A -85,B 0,C 180,E1 -833.404,E2 -833.404} C_VEL
LIN {X 0,Y 601.648,Z 676.219,A -85,B 0,C 180,E1 -836.081,E2 -836.081} C_VEL
LIN {X 0,Y 601.694,Z 661.934,A -85,B 0,C 180,E1 -838.833,E2 -838.833} C_VEL
LIN {X 0,Y 601.791,Z 647.413,A -85,B 0,C 180,E1 -841.703,E2 -841.703} C_VEL
LIN {X 0,Y 601.831,Z 634.646,A -85,B 0,C 180,E1 -844.294,E2 -844.294} C_VEL
LIN {X 0,Y 601.749,Z 627.248,A -85,B 0,C 180,E1 -845.729,E2 -845.729} C_VEL
LIN {X 0,Y 601.414,Z 625.57,A -85,B 0,C 180,E1 -846.112,E2 -846.112} C_VEL
LIN {X 0,Y 601.434,Z 625.566,A -85,B 0,C 180,E1 -848.471,E2 -848.471} C_VEL
LIN {X 0,Y 601.414,Z 625.575,A -85,B 0,C 180,E1 -850.874,E2 -850.874} C_VEL
LIN {X 0,Y 601.426,Z 625.564,A -85,B 0,C 180,E1 -853.585,E2 -853.585} C_VEL
LIN {X 0,Y 601.448,Z 625.569,A -85,B 0,C 180,E1 -856.424,E2 -856.424} C_VEL
LIN {X 0,Y 601.416,Z 625.565,A -85,B 0,C 180,E1 -859.426,E2 -859.426} C_VEL
LIN {X 0,Y 601.426,Z 625.566,A -85,B 0,C 180,E1 -861.732,E2 -861.732} C_VEL
LIN {X 0,Y 601.402,Z 625.575,A -85,B 0,C 180,E1 -864.246,E2 -864.246} C_VEL
LIN {X 0,Y 601.422,Z 625.565,A -85,B 0,C 180,E1 -866.686,E2 -866.686} C_VEL
LIN {X 0,Y 601.429,Z 625.563,A -85,B 0,C 180,E1 -869.058,E2 -869.058} C_VEL
LIN {X 0,Y 601.425,Z 625.567,A -85,B 0,C 180,E1 -871.373,E2 -871.373} C_VEL
LIN {X 0,Y 601.404,Z 625.576,A -85,B 0,C 180,E1 -873.636,E2 -873.636} C_VEL
LIN {X 0,Y 601.417,Z 625.565,A -85,B 0,C 180,E1 -876.589,E2 -876.589} C_VEL
LIN {X 0,Y 601.433,Z 625.57,A -85,B 0,C 180,E1 -879.478,E2 -879.478} C_VEL
LIN {X 0,Y 601.395,Z 625.567,A -85,B 0,C 180,E1 -882.311,E2 -882.311} C_VEL
LIN {X 0,Y 601.413,Z 625.566,A -85,B 0,C 180,E1 -884.409,E2 -884.409} C_VEL
LIN {X 0,Y 601.422,Z 625.57,A -85,B 0,C 180,E1 -887.172,E2 -887.172} C_VEL
LIN {X 0,Y 601.432,Z 625.563,A -85,B 0,C 180,E1 -889.905,E2 -889.905} C_VEL
LIN {X 0,Y 601.436,Z 625.572,A -85,B 0,C 180,E1 -892.615,E2 -892.615} C_VEL
LIN {X 0,Y 601.431,Z 625.563,A -85,B 0,C 180,E1 -895.308,E2 -895.308} C_VEL
LIN {X 0,Y 601.418,Z 625.569,A -85,B 0,C 180,E1 -897.991,E2 -897.991} C_VEL
LIN {X 0,Y 601.448,Z 625.564,A -85,B 0,C 180,E1 -900.669,E2 -900.669} C_VEL
LIN {X 0,Y 601.426,Z 625.565,A -85,B 0,C 180,E1 -903.349,E2 -903.349} C_VEL
LIN {X 0,Y 601.472,Z 625.761,A -85,B 0,C 180,E1 -905.448,E2 -905.448} C_VEL
LIN {X 0,Y 601.652,Z 634.349,A -85,B 0,C 180,E1 -907.382,E2 -907.382} C_VEL
LIN {X 0,Y 601.636,Z 644.853,A -85,B 0,C 180,E1 -910.092,E2 -910.092} C_VEL
LIN {X 0,Y 601.589,Z 652.137,A -85,B 0,C 180,E1 -911.924,E2 -911.924} C_VEL
LIN {X 0,Y 600.908,Z 654.357,A -85,B 0,C 180,E1 -912.441,E2 -912.441} C_VEL
LIN {X 0,Y 595.198,Z 662.219,A -85,B 0,C 180,E1 -914.102,E2 -914.102} C_VEL
LIN {X 0,Y 594.539,Z 664.474,A -85,B 0,C 180,E1 -914.627,E2 -914.627} C_VEL
LIN {X 0,Y 594.488,Z 674.999,A -85,B 0,C 180,E1 -917.19,E2 -917.19} C_VEL
LIN {X 0,Y 594.466,Z 685.461,A -85,B 0,C 180,E1 -919.69,E2 -919.69} C_VEL
LIN {X 0,Y 594.409,Z 696.283,A -85,B 0,C 180,E1 -922.232,E2 -922.232} C_VEL
LIN {X 0,Y 594.374,Z 707.467,A -85,B 0,C 180,E1 -924.819,E2 -924.819} C_VEL
LIN {X 0,Y 594.328,Z 720.731,A -85,B 0,C 180,E1 -927.845,E2 -927.845} C_VEL
LIN {X 0,Y 594.311,Z 725.77,A -85,B 0,C 180,E1 -928.974,E2 -928.974} C_VEL
LIN {X 0,Y 594.657,Z 731.913,A -85,B 0,C 180,E1 -929.081,E2 -929.081} C_VEL
LIN {X 0,Y 594.618,Z 745.069,A -85,B 0,C 180,E1 -929.398,E2 -929.398} C_VEL
LIN {X 0,Y 594.574,Z 757.829,A -85,B 0,C 180,E1 -929.854,E2 -929.854} C_VEL
LIN {X 0,Y 594.514,Z 769.242,A -85,B 0,C 180,E1 -930.402,E2 -930.402} C_VEL
LIN {X 0,Y 594.481,Z 779.857,A -85,B 0,C 180,E1 -931.047,E2 -931.047} C_VEL
LIN {X 0,Y 594.405,Z 790.721,A -85,B 0,C 180,E1 -931.867,E2 -931.867} C_VEL
LIN {X 0,Y 594.354,Z 799.901,A -85,B 0,C 180,E1 -932.728,E2 -932.728} C_VEL
LIN {X 0,Y 594.33,Z 808.872,A -85,B 0,C 180,E1 -933.764,E2 -933.764} C_VEL
LIN {X 0,Y 594.302,Z 815.863,A -85,B 0,C 180,E1 -934.768,E2 -934.768} C_VEL
LIN {X 0,Y 594.286,Z 821.768,A -85,B 0,C 180,E1 -935.83,E2 -935.83} C_VEL
LIN {X 0,Y 594.24,Z 827.119,A -85,B 0,C 180,E1 -937.097,E2 -937.097} C_VEL
LIN {X 0,Y 594.267,Z 829.81,A -85,B 0,C 180,E1 -937.95,E2 -937.95} C_VEL
LIN {X 0,Y 594.234,Z 831.843,A -85,B 0,C 180,E1 -938.817,E2 -938.817} C_VEL
LIN {X 0,Y 594.227,Z 833.263,A -85,B 0,C 180,E1 -939.758,E2 -939.758} C_VEL
LIN {X 0,Y 594.214,Z 833.951,A -85,B 0,C 180,E1 -940.805,E2 -940.805} C_VEL
LIN {X 0,Y 594.245,Z 833.707,A -85,B 0,C 180,E1 -941.835,E2 -941.835} C_VEL
LIN {X 0,Y 594.246,Z 832.586,A -85,B 0,C 180,E1 -942.841,E2 -942.841} C_VEL
LIN {X 0,Y 594.244,Z 829.523,A -85,B 0,C 180,E1 -944.249,E2 -944.249} C_VEL
LIN {X 0,Y 594.269,Z 825.274,A -85,B 0,C 180,E1 -945.477,E2 -945.477} C_VEL
LIN {X 0,Y 594.301,Z 819.501,A -85,B 0,C 180,E1 -946.695,E2 -946.695} C_VEL
LIN {X 0,Y 594.308,Z 812.949,A -85,B 0,C 180,E1 -947.768,E2 -947.768} C_VEL
LIN {X 0,Y 594.323,Z 805.808,A -85,B 0,C 180,E1 -948.707,E2 -948.707} C_VEL
LIN {X 0,Y 594.364,Z 797.069,A -85,B 0,C 180,E1 -949.646,E2 -949.646} C_VEL
LIN {X 0,Y 594.437,Z 786.753,A -85,B 0,C 180,E1 -950.545,E2 -950.545} C_VEL
LIN {X 0,Y 594.486,Z 776.188,A -85,B 0,C 180,E1 -951.283,E2 -951.283} C_VEL
LIN {X 0,Y 594.516,Z 763.881,A -85,B 0,C 180,E1 -951.962,E2 -951.962} C_VEL
LIN {X 0,Y 594.603,Z 752.406,A -85,B 0,C 180,E1 -952.448,E2 -952.448} C_VEL
LIN {X 0,Y 594.661,Z 739.261,A -85,B 0,C 180,E1 -952.85,E2 -952.85} C_VEL
LIN {X 0,Y 594.518,Z 727.161,A -85,B 0,C 180,E1 -953.092,E2 -953.092} C_VEL
LIN {X 0,Y 594.306,Z 725.71,A -85,B 0,C 180,E1 -953.119,E2 -953.119} C_VEL
LIN {X 0,Y 594.334,Z 713.594,A -85,B 0,C 180,E1 -955.868,E2 -955.868} C_VEL
LIN {X 0,Y 594.39,Z 701.48,A -85,B 0,C 180,E1 -958.652,E2 -958.652} C_VEL
LIN {X 0,Y 594.445,Z 689.678,A -85,B 0,C 180,E1 -961.404,E2 -961.404} C_VEL
LIN {X 0,Y 594.495,Z 676.914,A -85,B 0,C 180,E1 -964.438,E2 -964.438} C_VEL
LIN {X 0,Y 594.554,Z 666.187,A -85,B 0,C 180,E1 -967.041,E2 -967.041} C_VEL
LIN {X 0,Y 594.626,Z 654.451,A -85,B 0,C 180,E1 -969.956,E2 -969.956} C_VEL
LIN {X 0,Y 594.701,Z 643.244,A -85,B 0,C 180,E1 -972.816,E2 -972.816} C_VEL
LIN {X 0,Y 594.684,Z 634.807,A -85,B 0,C 180,E1 -974.931,E2 -974.931} C_VEL
LIN {X 0,Y 594.408,Z 626.446,A -85,B 0,C 180,E1 -976.931,E2 -976.931} C_VEL
LIN {X 0,Y 594.396,Z 626.446,A -85,B 0,C 180,E1 -979.785,E2 -979.785} C_VEL
LIN {X 0,Y 594.397,Z 626.446,A -85,B 0,C 180,E1 -982.527,E2 -982.527} C_VEL
LIN {X 0,Y 594.4,Z 626.447,A -85,B 0,C 180,E1 -985.253,E2 -985.253} C_VEL
LIN {X 0,Y 594.405,Z 626.447,A -85,B 0,C 180,E1 -987.968,E2 -987.968} C_VEL
LIN {X 0,Y 594.428,Z 626.444,A -85,B 0,C 180,E1 -990.678,E2 -990.678} C_VEL
LIN {X 0,Y 594.387,Z 626.45,A -85,B 0,C 180,E1 -993.39,E2 -993.39} C_VEL
LIN {X 0,Y 594.364,Z 626.452,A -85,B 0,C 180,E1 -996.109,E2 -996.109} C_VEL
LIN {X 0,Y 594.403,Z 626.447,A -85,B 0,C 180,E1 -998.842,E2 -998.842} C_VEL
LIN {X 0,Y 594.398,Z 626.446,A -85,B 0,C 180,E1 -1001.596,E2 -1001.596} C_VEL
LIN {X 0,Y 594.391,Z 626.446,A -85,B 0,C 180,E1 -1004.377,E2 -1004.377} C_VEL
LIN {X 0,Y 594.396,Z 626.445,A -85,B 0,C 180,E1 -1007.193,E2 -1007.193} C_VEL
LIN {X 0,Y 594.376,Z 626.447,A -85,B 0,C 180,E1 -1010.054,E2 -1010.054} C_VEL
LIN {X 0,Y 594.364,Z 626.45,A -85,B 0,C 180,E1 -1012.967,E2 -1012.967} C_VEL
LIN {X 0,Y 594.376,Z 626.447,A -85,B 0,C 180,E1 -1015.193,E2 -1015.193} C_VEL
LIN {X 0,Y 594.412,Z 626.503,A -85,B 0,C 180,E1 -1016.44,E2 -1016.44} C_VEL
LIN {X 0,Y 594.542,Z 637.306,A -85,B 0,C 180,E1 -1016.834,E2 -1016.834} C_VEL
LIN {X 0,Y 594.509,Z 648.43,A -85,B 0,C 180,E1 -1017.359,E2 -1017.359} C_VEL
LIN {X 0,Y 594.438,Z 659.692,A -85,B 0,C 180,E1 -1018.035,E2 -1018.035} C_VEL
LIN {X 0,Y 594.426,Z 671.07,A -85,B 0,C 180,E1 -1018.898,E2 -1018.898} C_VEL
LIN {X 0,Y 594.344,Z 680.368,A -85,B 0,C 180,E1 -1019.778,E2 -1019.778} C_VEL
LIN {X 0,Y 594.327,Z 688.814,A -85,B 0,C 180,E1 -1020.76,E2 -1020.76} C_VEL
LIN {X 0,Y 594.298,Z 696.454,A -85,B 0,C 180,E1 -1021.865,E2 -1021.865} C_VEL
LIN {X 0,Y 594.261,Z 702.378,A -85,B 0,C 180,E1 -1022.958,E2 -1022.958} C_VEL
LIN {X 0,Y 594.264,Z 707.212,A -85,B 0,C 180,E1 -1024.122,E2 -1024.122} C_VEL
LIN {X 0,Y 594.224,Z 710.985,A -85,B 0,C 180,E1 -1025.418,E2 -1025.418} C_VEL
LIN {X 0,Y 594.221,Z 712.9,A -85,B 0,C 180,E1 -1026.462,E2 -1026.462} C_VEL
LIN {X 0,Y 594.227,Z 713.891,A -85,B 0,C 180,E1 -1027.588,E2 -1027.588} C_VEL
LIN {X 0,Y 594.208,Z 713.719,A -85,B 0,C 180,E1 -1028.819,E2 -1028.819} C_VEL
LIN {X 0,Y 594.227,Z 712.723,A -85,B 0,C 180,E1 -1029.757,E2 -1029.757} C_VEL
LIN {X 0,Y 594.23,Z 710.681,A -85,B 0,C 180,E1 -1030.806,E2 -1030.806} C_VEL
LIN {X 0,Y 594.262,Z 706.784,A -85,B 0,C 180,E1 -1032.086,E2 -1032.086} C_VEL
LIN {X 0,Y 594.274,Z 701.538,A -85,B 0,C 180,E1 -1033.308,E2 -1033.308} C_VEL
LIN {X 0,Y 594.308,Z 696.346,A -85,B 0,C 180,E1 -1034.243,E2 -1034.243} C_VEL
LIN {X 0,Y 594.309,Z 688.748,A -85,B 0,C 180,E1 -1035.339,E2 -1035.339} C_VEL
LIN {X 0,Y 594.345,Z 680.504,A -85,B 0,C 180,E1 -1036.297,E2 -1036.297} C_VEL
LIN {X 0,Y 594.385,Z 670.637,A -85,B 0,C 180,E1 -1037.231,E2 -1037.231} C_VEL
LIN {X 0,Y 594.477,Z 659.336,A -85,B 0,C 180,E1 -1038.078,E2 -1038.078} C_VEL
LIN {X 0,Y 594.503,Z 648.723,A -85,B 0,C 180,E1 -1038.716,E2 -1038.716} C_VEL
LIN {X 0,Y 594.545,Z 638.076,A -85,B 0,C 180,E1 -1039.223,E2 -1039.223} C_VEL
LIN {X 0,Y 594.593,Z 627.601,A -85,B 0,C 180,E1 -1039.611,E2 -1039.611} C_VEL
LIN {X 0,Y 594.405,Z 626.446,A -85,B 0,C 180,E1 -1039.675,E2 -1039.675} C_VEL
LIN {X 0,Y 594.392,Z 626.439,A -85,B 0,C 180,E1 -1042.391,E2 -1042.391} C_VEL
LIN {X 0,Y 594.383,Z 626.448,A -85,B 0,C 180,E1 -1045.42,E2 -1045.42} C_VEL
LIN {X 0,Y 594.379,Z 626.441,A -85,B 0,C 180,E1 -1048.357,E2 -1048.357} C_VEL
LIN {X 0,Y 594.385,Z 626.441,A -85,B 0,C 180,E1 -1051.042,E2 -1051.042} C_VEL
LIN {X 0,Y 594.387,Z 626.445,A -85,B 0,C 180,E1 -1053.977,E2 -1053.977} C_VEL
LIN {X 0,Y 594.389,Z 626.441,A -85,B 0,C 180,E1 -1056.296,E2 -1056.296} C_VEL
LIN {X 0,Y 594.408,Z 626.439,A -85,B 0,C 180,E1 -1059.225,E2 -1059.225} C_VEL
LIN {X 0,Y 594.354,Z 626.449,A -85,B 0,C 180,E1 -1062.095,E2 -1062.095} C_VEL
LIN {X 0,Y 594.367,Z 626.446,A -85,B 0,C 180,E1 -1064.219,E2 -1064.219} C_VEL
LIN {X 0,Y 594.38,Z 626.444,A -85,B 0,C 180,E1 -1066.321,E2 -1066.321} C_VEL
LIN {X 0,Y 594.379,Z 626.44,A -85,B 0,C 180,E1 -1069.095,E2 -1069.095} C_VEL
LIN {X 0,Y 594.421,Z 626.444,A -85,B 0,C 180,E1 -1071.843,E2 -1071.843} C_VEL
LIN {X 0,Y 594.388,Z 626.441,A -85,B 0,C 180,E1 -1074.572,E2 -1074.572} C_VEL
LIN {X 0,Y 594.413,Z 626.436,A -85,B 0,C 180,E1 -1077.289,E2 -1077.289} C_VEL
LIN {X 0,Y 594.417,Z 626.445,A -85,B 0,C 180,E1 -1080,E2 -1080} C_VEL
LIN {X 0,Y 594.413,Z 626.438,A -85,B 0,C 180,E1 -1082.711,E2 -1082.711} C_VEL
LIN {X 0,Y 594.388,Z 626.439,A -85,B 0,C 180,E1 -1085.428,E2 -1085.428} C_VEL
LIN {X 0,Y 594.421,Z 626.446,A -85,B 0,C 180,E1 -1088.157,E2 -1088.157} C_VEL
LIN {X 0,Y 594.391,Z 626.439,A -85,B 0,C 180,E1 -1091.074,E2 -1091.074} C_VEL
LIN {X 0,Y 594.381,Z 626.441,A -85,B 0,C 180,E1 -1093.679,E2 -1093.679} C_VEL
LIN {X 0,Y 594.397,Z 626.442,A -85,B 0,C 180,E1 -1096.72,E2 -1096.72} C_VEL
LIN {X 0,Y 594.368,Z 626.441,A -85,B 0,C 180,E1 -1099.335,E2 -1099.335} C_VEL
LIN {X 0,Y 594.367,Z 626.442,A -85,B 0,C 180,E1 -1101.503,E2 -1101.503} C_VEL
LIN {X 0,Y 594.391,Z 626.449,A -85,B 0,C 180,E1 -1104.446,E2 -1104.446} C_VEL
LIN {X 0,Y 594.386,Z 626.446,A -85,B 0,C 180,E1 -1106.7,E2 -1106.7} C_VEL
LIN {X 0,Y 594.384,Z 626.442,A -85,B 0,C 180,E1 -1108.999,E2 -1108.999} C_VEL
LIN {X 0,Y 594.379,Z 626.44,A -85,B 0,C 180,E1 -1111.643,E2 -1111.643} C_VEL
LIN {X 0,Y 594.381,Z 626.451,A -85,B 0,C 180,E1 -1114.58,E2 -1114.58} C_VEL
LIN {X 0,Y 594.393,Z 626.439,A -85,B 0,C 180,E1 -1117.609,E2 -1117.609} C_VEL
LIN {X 0,Y 594.374,Z 626.451,A -85,B 0,C 180,E1 -1120.567,E2 -1120.567} C_VEL
LIN {X 0,Y 594.383,Z 626.441,A -85,B 0,C 180,E1 -1123.298,E2 -1123.298} C_VEL
LIN {X 0,Y 594.363,Z 626.445,A -85,B 0,C 180,E1 -1126.161,E2 -1126.161} C_VEL
LIN {X 0,Y 594.383,Z 626.448,A -85,B 0,C 180,E1 -1128.536,E2 -1128.536} C_VEL
LIN {X 0,Y 594.379,Z 626.445,A -85,B 0,C 180,E1 -1131.297,E2 -1131.297} C_VEL
LIN {X 0,Y 594.389,Z 626.518,A -85,B 0,C 180,E1 -1133.784,E2 -1133.784} C_VEL
LIN {X 0,Y 594.877,Z 630.764,A -85,B 0,C 180,E1 -1134.627,E2 -1134.627} C_VEL
LIN {X 0,Y 594.953,Z 643.496,A -85,B 0,C 180,E1 -1137.086,E2 -1137.086} C_VEL
LIN {X 0,Y 594.854,Z 657.501,A -85,B 0,C 180,E1 -1139.921,E2 -1139.921} C_VEL
LIN {X 0,Y 594.746,Z 670.886,A -85,B 0,C 180,E1 -1142.558,E2 -1142.558} C_VEL
LIN {X 0,Y 594.654,Z 684.582,A -85,B 0,C 180,E1 -1145.193,E2 -1145.193} C_VEL
LIN {X 0,Y 594.575,Z 700.232,A -85,B 0,C 180,E1 -1148.14,E2 -1148.14} C_VEL
LIN {X 0,Y 594.492,Z 715.954,A -85,B 0,C 180,E1 -1151.041,E2 -1151.041} C_VEL
LIN {X 0,Y 594.419,Z 731.534,A -85,B 0,C 180,E1 -1153.868,E2 -1153.868} C_VEL
LIN {X 0,Y 594.365,Z 747.185,A -85,B 0,C 180,E1 -1156.669,E2 -1156.669} C_VEL
LIN {X 0,Y 594.353,Z 754.155,A -85,B 0,C 180,E1 -1157.906,E2 -1157.906} C_VEL
LIN {X 0,Y 594.67,Z 759.932,A -85,B 0,C 180,E1 -1157.999,E2 -1157.999} C_VEL
LIN {X 0,Y 594.627,Z 773.205,A -85,B 0,C 180,E1 -1158.301,E2 -1158.301} C_VEL
LIN {X 0,Y 594.562,Z 786.294,A -85,B 0,C 180,E1 -1158.746,E2 -1158.746} C_VEL
LIN {X 0,Y 594.518,Z 797.628,A -85,B 0,C 180,E1 -1159.269,E2 -1159.269} C_VEL
LIN {X 0,Y 594.47,Z 809.195,A -85,B 0,C 180,E1 -1159.957,E2 -1159.957} C_VEL
LIN {X 0,Y 594.414,Z 819.591,A -85,B 0,C 180,E1 -1160.729,E2 -1160.729} C_VEL
LIN {X 0,Y 594.383,Z 828.109,A -85,B 0,C 180,E1 -1161.5,E2 -1161.5} C_VEL
LIN {X 0,Y 594.347,Z 835.958,A -85,B 0,C 180,E1 -1162.355,E2 -1162.355} C_VEL
LIN {X 0,Y 594.283,Z 843.811,A -85,B 0,C 180,E1 -1163.408,E2 -1163.408} C_VEL
LIN {X 0,Y 594.289,Z 850.679,A -85,B 0,C 180,E1 -1164.571,E2 -1164.571} C_VEL
LIN {X 0,Y 594.271,Z 855.37,A -85,B 0,C 180,E1 -1165.591,E2 -1165.591} C_VEL
LIN {X 0,Y 594.268,Z 858.955,A -85,B 0,C 180,E1 -1166.61,E2 -1166.61} C_VEL
LIN {X 0,Y 594.226,Z 860.809,A -85,B 0,C 180,E1 -1167.288,E2 -1167.288} C_VEL
LIN {X 0,Y 594.239,Z 862.201,A -85,B 0,C 180,E1 -1167.966,E2 -1167.966} C_VEL
LIN {X 0,Y 594.239,Z 863.784,A -85,B 0,C 180,E1 -1169.322,E2 -1169.322} C_VEL
LIN {X 0,Y 594.236,Z 864,A -85,B 0,C 180,E1 -1170,E2 -1170} C_VEL
LIN {X 0,Y 594.247,Z 863.185,A -85,B 0,C 180,E1 -1171.355,E2 -1171.355} C_VEL
LIN {X 0,Y 594.239,Z 862.202,A -85,B 0,C 180,E1 -1172.033,E2 -1172.033} C_VEL
LIN {X 0,Y 594.226,Z 860.81,A -85,B 0,C 180,E1 -1172.711,E2 -1172.711} C_VEL
LIN {X 0,Y 594.289,Z 857.897,A -85,B 0,C 180,E1 -1173.729,E2 -1173.729} C_VEL
LIN {X 0,Y 594.241,Z 853.952,A -85,B 0,C 180,E1 -1174.748,E2 -1174.748} C_VEL
LIN {X 0,Y 594.304,Z 847.879,A -85,B 0,C 180,E1 -1175.939,E2 -1175.939} C_VEL
LIN {X 0,Y 594.308,Z 841.239,A -85,B 0,C 180,E1 -1176.962,E2 -1176.962} C_VEL
LIN {X 0,Y 594.359,Z 832.993,A -85,B 0,C 180,E1 -1177.986,E2 -1177.986} C_VEL
LIN {X 0,Y 594.382,Z 824.542,A -85,B 0,C 180,E1 -1178.842,E2 -1178.842} C_VEL
LIN {X 0,Y 594.429,Z 814.099,A -85,B 0,C 180,E1 -1179.699,E2 -1179.699} C_VEL
LIN {X 0,Y 594.488,Z 803.765,A -85,B 0,C 180,E1 -1180.386,E2 -1180.386} C_VEL
LIN {X 0,Y 594.547,Z 792.84,A -85,B 0,C 180,E1 -1180.968,E2 -1180.968} C_VEL
LIN {X 0,Y 594.6,Z 780.758,A -85,B 0,C 180,E1 -1181.462,E2 -1181.462} C_VEL
LIN {X 0,Y 594.651,Z 767.373,A -85,B 0,C 180,E1 -1181.85,E2 -1181.85} C_VEL
LIN {X 0,Y 594.574,Z 755.633,A -85,B 0,C 180,E1 -1182.067,E2 -1182.067} C_VEL
LIN {X 0,Y 594.358,Z 754.037,A -85,B 0,C 180,E1 -1182.115,E2 -1182.115} C_VEL
LIN {X 0,Y 594.395,Z 739.364,A -85,B 0,C 180,E1 -1184.726,E2 -1184.726} C_VEL
LIN {X 0,Y 594.466,Z 723.713,A -85,B 0,C 180,E1 -1187.545,E2 -1187.545} C_VEL
LIN {X 0,Y 594.527,Z 708.061,A -85,B 0,C 180,E1 -1190.409,E2 -1190.409} C_VEL
LIN {X 0,Y 594.614,Z 694.367,A -85,B 0,C 180,E1 -1192.956,E2 -1192.956} C_VEL
LIN {X 0,Y 594.696,Z 680.672,A -85,B 0,C 180,E1 -1195.553,E2 -1195.553} C_VEL
LIN {X 0,Y 594.789,Z 665.021,A -85,B 0,C 180,E1 -1198.59,E2 -1198.59} C_VEL
LIN {X 0,Y 594.895,Z 651.326,A -85,B 0,C 180,E1 -1201.319,E2 -1201.319} C_VEL
LIN {X 0,Y 594.939,Z 639.369,A -85,B 0,C 180,E1 -1203.724,E2 -1203.724} C_VEL
LIN {X 0,Y 594.856,Z 628.869,A -85,B 0,C 180,E1 -1205.789,E2 -1205.789} C_VEL
LIN {X 0,Y 594.402,Z 626.445,A -85,B 0,C 180,E1 -1206.331,E2 -1206.331} C_VEL
LIN {X 0,Y 594.388,Z 626.449,A -85,B 0,C 180,E1 -1208.804,E2 -1208.804} C_VEL
LIN {X 0,Y 594.379,Z 626.442,A -85,B 0,C 180,E1 -1211.848,E2 -1211.848} C_VEL
LIN {X 0,Y 594.361,Z 626.451,A -85,B 0,C 180,E1 -1214.808,E2 -1214.808} C_VEL
LIN {X 0,Y 594.369,Z 626.443,A -85,B 0,C 180,E1 -1217.624,E2 -1217.624} C_VEL
LIN {X 0,Y 594.394,Z 626.449,A -85,B 0,C 180,E1 -1220.321,E2 -1220.321} C_VEL
LIN {X 0,Y 594.385,Z 626.442,A -85,B 0,C 180,E1 -1222.913,E2 -1222.913} C_VEL
LIN {X 0,Y 594.378,Z 626.448,A -85,B 0,C 180,E1 -1225.861,E2 -1225.861} C_VEL
LIN {X 0,Y 594.386,Z 626.441,A -85,B 0,C 180,E1 -1228.651,E2 -1228.651} C_VEL
LIN {X 0,Y 594.378,Z 626.442,A -85,B 0,C 180,E1 -1231.042,E2 -1231.042} C_VEL
LIN {X 0,Y 594.385,Z 626.445,A -85,B 0,C 180,E1 -1233.976,E2 -1233.976} C_VEL
LIN {X 0,Y 594.389,Z 626.441,A -85,B 0,C 180,E1 -1236.296,E2 -1236.296} C_VEL
LIN {X 0,Y 594.405,Z 626.446,A -85,B 0,C 180,E1 -1239.224,E2 -1239.224} C_VEL
LIN {X 0,Y 594.377,Z 626.442,A -85,B 0,C 180,E1 -1242.096,E2 -1242.096} C_VEL
LIN {X 0,Y 594.365,Z 626.443,A -85,B 0,C 180,E1 -1244.219,E2 -1244.219} C_VEL
LIN {X 0,Y 594.369,Z 626.452,A -85,B 0,C 180,E1 -1247.017,E2 -1247.017} C_VEL
LIN {X 0,Y 594.392,Z 626.44,A -85,B 0,C 180,E1 -1249.784,E2 -1249.784} C_VEL
LIN {X 0,Y 594.389,Z 626.448,A -85,B 0,C 180,E1 -1252.527,E2 -1252.527} C_VEL
LIN {X 0,Y 594.398,Z 626.44,A -85,B 0,C 180,E1 -1255.252,E2 -1255.252} C_VEL
LIN {X 0,Y 594.389,Z 626.444,A -85,B 0,C 180,E1 -1257.967,E2 -1257.967} C_VEL
LIN {X 0,Y 594.419,Z 626.44,A -85,B 0,C 180,E1 -1260.677,E2 -1260.677} C_VEL
LIN {X 0,Y 594.379,Z 626.443,A -85,B 0,C 180,E1 -1263.389,E2 -1263.389} C_VEL
LIN {X 0,Y 594.415,Z 626.485,A -85,B 0,C 180,E1 -1265.342,E2 -1265.342} C_VEL
LIN {X 0,Y 594.677,Z 637.401,A -85,B 0,C 180,E1 -1267.811,E2 -1267.811} C_VEL
LIN {X 0,Y 594.677,Z 646.88,A -85,B 0,C 180,E1 -1270.211,E2 -1270.211} C_VEL
LIN {X 0,Y 594.61,Z 657.814,A -85,B 0,C 180,E1 -1272.978,E2 -1272.978} C_VEL
LIN {X 0,Y 594.539,Z 664.474,A -85,B 0,C 180,E1 -1274.627,E2 -1274.627} C_VEL
LIN {X 0,Y 593.869,Z 666.727,A -85,B 0,C 180,E1 -1275.149,E2 -1275.149} C_VEL
LIN {X 0,Y 588.13,Z 674.638,A -85,B 0,C 180,E1 -1276.828,E2 -1276.828} C_VEL
LIN {X 0,Y 587.501,Z 676.92,A -85,B 0,C 180,E1 -1277.358,E2 -1277.358} C_VEL
LIN {X 0,Y 587.443,Z 689.128,A -85,B 0,C 180,E1 -1280.301,E2 -1280.301} C_VEL
LIN {X 0,Y 587.378,Z 701.629,A -85,B 0,C 180,E1 -1283.256,E2 -1283.256} C_VEL
LIN {X 0,Y 587.291,Z 714.153,A -85,B 0,C 180,E1 -1286.169,E2 -1286.169} C_VEL
LIN {X 0,Y 587.249,Z 725.653,A -85,B 0,C 180,E1 -1288.811,E2 -1288.811} C_VEL
LIN {X 0,Y 587.727,Z 731.207,A -85,B 0,C 180,E1 -1288.924,E2 -1288.924} C_VEL
LIN {X 0,Y 587.684,Z 744.896,A -85,B 0,C 180,E1 -1289.253,E2 -1289.253} C_VEL
LIN {X 0,Y 587.616,Z 757.581,A -85,B 0,C 180,E1 -1289.709,E2 -1289.709} C_VEL
LIN {X 0,Y 587.513,Z 769.525,A -85,B 0,C 180,E1 -1290.29,E2 -1290.29} C_VEL
LIN {X 0,Y 587.455,Z 780.348,A -85,B 0,C 180,E1 -1290.959,E2 -1290.959} C_VEL
LIN {X 0,Y 587.378,Z 790.845,A -85,B 0,C 180,E1 -1291.767,E2 -1291.767} C_VEL
LIN {X 0,Y 587.332,Z 799.45,A -85,B 0,C 180,E1 -1292.579,E2 -1292.579} C_VEL
LIN {X 0,Y 587.254,Z 808.334,A -85,B 0,C 180,E1 -1293.607,E2 -1293.607} C_VEL
LIN {X 0,Y 587.235,Z 815.733,A -85,B 0,C 180,E1 -1294.671,E2 -1294.671} C_VEL
LIN {X 0,Y 587.202,Z 820.554,A -85,B 0,C 180,E1 -1295.526,E2 -1295.526} C_VEL
LIN {X 0,Y 587.191,Z 826.072,A -85,B 0,C 180,E1 -1296.758,E2 -1296.758} C_VEL
LIN {X 0,Y 587.154,Z 829.561,A -85,B 0,C 180,E1 -1297.816,E2 -1297.816} C_VEL
LIN {X 0,Y 587.152,Z 832.094,A -85,B 0,C 180,E1 -1298.921,E2 -1298.921} C_VEL
LIN {X 0,Y 587.135,Z 833.723,A -85,B 0,C 180,E1 -1300.269,E2 -1300.269} C_VEL
LIN {X 0,Y 587.119,Z 833.977,A -85,B 0,C 180,E1 -1301.175,E2 -1301.175} C_VEL
LIN {X 0,Y 587.158,Z 833.539,A -85,B 0,C 180,E1 -1302.09,E2 -1302.09} C_VEL
LIN {X 0,Y 587.144,Z 832.203,A -85,B 0,C 180,E1 -1303.101,E2 -1303.101} C_VEL
LIN {X 0,Y 587.158,Z 828.926,A -85,B 0,C 180,E1 -1304.486,E2 -1304.486} C_VEL
LIN {X 0,Y 587.188,Z 825.34,A -85,B 0,C 180,E1 -1305.515,E2 -1305.515} C_VEL
LIN {X 0,Y 587.22,Z 819.747,A -85,B 0,C 180,E1 -1306.717,E2 -1306.717} C_VEL
LIN {X 0,Y 587.255,Z 812.457,A -85,B 0,C 180,E1 -1307.92,E2 -1307.92} C_VEL
LIN {X 0,Y 587.277,Z 804.685,A -85,B 0,C 180,E1 -1308.932,E2 -1308.932} C_VEL
LIN {X 0,Y 587.365,Z 795.601,A -85,B 0,C 180,E1 -1309.892,E2 -1309.892} C_VEL
LIN {X 0,Y 587.393,Z 785.445,A -85,B 0,C 180,E1 -1310.761,E2 -1310.761} C_VEL
LIN {X 0,Y 587.475,Z 774.154,A -85,B 0,C 180,E1 -1311.533,E2 -1311.533} C_VEL
LIN {X 0,Y 587.531,Z 763.009,A -85,B 0,C 180,E1 -1312.138,E2 -1312.138} C_VEL
LIN {X 0,Y 587.655,Z 751.106,A -85,B 0,C 180,E1 -1312.632,E2 -1312.632} C_VEL
LIN {X 0,Y 587.719,Z 737.803,A -85,B 0,C 180,E1 -1313.027,E2 -1313.027} C_VEL
LIN {X 0,Y 587.62,Z 728.242,A -85,B 0,C 180,E1 -1313.22,E2 -1313.22} C_VEL
LIN {X 0,Y 587.236,Z 725.669,A -85,B 0,C 180,E1 -1313.276,E2 -1313.276} C_VEL
LIN {X 0,Y 587.284,Z 712.994,A -85,B 0,C 180,E1 -1316.189,E2 -1316.189} C_VEL
LIN {X 0,Y 587.352,Z 700.773,A -85,B 0,C 180,E1 -1319.035,E2 -1319.035} C_VEL
LIN {X 0,Y 587.422,Z 689.093,A -85,B 0,C 180,E1 -1321.799,E2 -1321.799} C_VEL
LIN {X 0,Y 587.486,Z 677.912,A -85,B 0,C 180,E1 -1324.491,E2 -1324.491} C_VEL
LIN {X 0,Y 587.565,Z 667.389,A -85,B 0,C 180,E1 -1327.075,E2 -1327.075} C_VEL
LIN {X 0,Y 587.651,Z 656.899,A -85,B 0,C 180,E1 -1329.707,E2 -1329.707} C_VEL
LIN {X 0,Y 587.752,Z 645.641,A -85,B 0,C 180,E1 -1332.607,E2 -1332.607} C_VEL
LIN {X 0,Y 587.699,Z 635.407,A -85,B 0,C 180,E1 -1335.102,E2 -1335.102} C_VEL
LIN {X 0,Y 587.39,Z 627.488,A -85,B 0,C 180,E1 -1336.992,E2 -1336.992} C_VEL
LIN {X 0,Y 587.344,Z 627.324,A -85,B 0,C 180,E1 -1339.661,E2 -1339.661} C_VEL
LIN {X 0,Y 587.369,Z 627.321,A -85,B 0,C 180,E1 -1342.437,E2 -1342.437} C_VEL
LIN {X 0,Y 587.369,Z 627.322,A -85,B 0,C 180,E1 -1345.196,E2 -1345.196} C_VEL
LIN {X 0,Y 587.375,Z 627.322,A -85,B 0,C 180,E1 -1347.943,E2 -1347.943} C_VEL
LIN {X 0,Y 587.399,Z 627.32,A -85,B 0,C 180,E1 -1350.686,E2 -1350.686} C_VEL
LIN {X 0,Y 587.339,Z 627.328,A -85,B 0,C 180,E1 -1353.43,E2 -1353.43} C_VEL
LIN {X 0,Y 587.357,Z 627.321,A -85,B 0,C 180,E1 -1355.493,E2 -1355.493} C_VEL
LIN {X 0,Y 587.374,Z 627.32,A -85,B 0,C 180,E1 -1358.255,E2 -1358.255} C_VEL
LIN {X 0,Y 587.351,Z 627.324,A -85,B 0,C 180,E1 -1361.134,E2 -1361.134} C_VEL
LIN {X 0,Y 587.368,Z 627.322,A -85,B 0,C 180,E1 -1364.261,E2 -1364.261} C_VEL
LIN {X 0,Y 587.362,Z 627.321,A -85,B 0,C 180,E1 -1367.406,E2 -1367.406} C_VEL
LIN {X 0,Y 587.331,Z 627.326,A -85,B 0,C 180,E1 -1370.305,E2 -1370.305} C_VEL
LIN {X 0,Y 587.322,Z 627.33,A -85,B 0,C 180,E1 -1373.259,E2 -1373.259} C_VEL
LIN {X 0,Y 587.337,Z 627.325,A -85,B 0,C 180,E1 -1375.517,E2 -1375.517} C_VEL
LIN {X 0,Y 587.343,Z 627.334,A -85,B 0,C 180,E1 -1376.326,E2 -1376.326} C_VEL
LIN {X 0,Y 587.617,Z 633.649,A -85,B 0,C 180,E1 -1376.552,E2 -1376.552} C_VEL
LIN {X 0,Y 587.548,Z 644.665,A -85,B 0,C 180,E1 -1377.036,E2 -1377.036} C_VEL
LIN {X 0,Y 587.494,Z 655.103,A -85,B 0,C 180,E1 -1377.617,E2 -1377.617} C_VEL
LIN {X 0,Y 587.438,Z 665,A -85,B 0,C 180,E1 -1378.299,E2 -1378.299} C_VEL
LIN {X 0,Y 587.331,Z 674.859,A -85,B 0,C 180,E1 -1379.13,E2 -1379.13} C_VEL
LIN {X 0,Y 587.286,Z 683.096,A -85,B 0,C 180,E1 -1379.975,E2 -1379.975} C_VEL
LIN {X 0,Y 587.253,Z 691.046,A -85,B 0,C 180,E1 -1380.971,E2 -1380.971} C_VEL
LIN {X 0,Y 587.21,Z 698.71,A -85,B 0,C 180,E1 -1382.181,E2 -1382.181} C_VEL
LIN {X 0,Y 587.167,Z 703.27,A -85,B 0,C 180,E1 -1383.086,E2 -1383.086} C_VEL
LIN {X 0,Y 587.157,Z 708.027,A -85,B 0,C 180,E1 -1384.32,E2 -1384.32} C_VEL
LIN {X 0,Y 587.137,Z 711.267,A -85,B 0,C 180,E1 -1385.516,E2 -1385.516} C_VEL
LIN {X 0,Y 587.124,Z 713.286,A -85,B 0,C 180,E1 -1386.763,E2 -1386.763} C_VEL
LIN {X 0,Y 587.119,Z 713.953,A -85,B 0,C 180,E1 -1387.811,E2 -1387.811} C_VEL
LIN {X 0,Y 587.113,Z 713.66,A -85,B 0,C 180,E1 -1388.915,E2 -1388.915} C_VEL
LIN {X 0,Y 587.144,Z 711.906,A -85,B 0,C 180,E1 -1390.269,E2 -1390.269} C_VEL
LIN {X 0,Y 587.136,Z 709.826,A -85,B 0,C 180,E1 -1391.174,E2 -1391.174} C_VEL
LIN {X 0,Y 587.191,Z 706.94,A -85,B 0,C 180,E1 -1392.092,E2 -1392.092} C_VEL
LIN {X 0,Y 587.198,Z 702.792,A -85,B 0,C 180,E1 -1393.106,E2 -1393.106} C_VEL
LIN {X 0,Y 587.22,Z 696.638,A -85,B 0,C 180,E1 -1394.269,E2 -1394.269} C_VEL
LIN {X 0,Y 587.257,Z 690.153,A -85,B 0,C 180,E1 -1395.243,E2 -1395.243} C_VEL
LIN {X 0,Y 587.279,Z 681.702,A -85,B 0,C 180,E1 -1396.267,E2 -1396.267} C_VEL
LIN {X 0,Y 587.354,Z 673.176,A -85,B 0,C 180,E1 -1397.114,E2 -1397.114} C_VEL
LIN {X 0,Y 587.442,Z 663.089,A -85,B 0,C 180,E1 -1397.935,E2 -1397.935} C_VEL
LIN {X 0,Y 587.477,Z 651.615,A -85,B 0,C 180,E1 -1398.684,E2 -1398.684} C_VEL
LIN {X 0,Y 587.591,Z 640.257,A -85,B 0,C 180,E1 -1399.262,E2 -1399.262} C_VEL
LIN {X 0,Y 587.625,Z 628.644,A -85,B 0,C 180,E1 -1399.715,E2 -1399.715} C_VEL
LIN {X 0,Y 587.362,Z 627.322,A -85,B 0,C 180,E1 -1399.789,E2 -1399.789} C_VEL
LIN {X 0,Y 587.348,Z 627.317,A -85,B 0,C 180,E1 -1402.393,E2 -1402.393} C_VEL
LIN {X 0,Y 587.364,Z 627.322,A -85,B 0,C 180,E1 -1405.78,E2 -1405.78} C_VEL
LIN {X 0,Y 587.344,Z 627.319,A -85,B 0,C 180,E1 -1408.231,E2 -1408.231} C_VEL
LIN {X 0,Y 587.351,Z 627.316,A -85,B 0,C 180,E1 -1410.866,E2 -1410.866} C_VEL
LIN {X 0,Y 587.36,Z 627.323,A -85,B 0,C 180,E1 -1413.819,E2 -1413.819} C_VEL
LIN {X 0,Y 587.337,Z 627.323,A -85,B 0,C 180,E1 -1415.994,E2 -1415.994} C_VEL
LIN {X 0,Y 587.322,Z 627.323,A -85,B 0,C 180,E1 -1418.226,E2 -1418.226} C_VEL
LIN {X 0,Y 587.35,Z 627.317,A -85,B 0,C 180,E1 -1421.151,E2 -1421.151} C_VEL
LIN {X 0,Y 587.326,Z 627.327,A -85,B 0,C 180,E1 -1424.025,E2 -1424.025} C_VEL
LIN {X 0,Y 587.358,Z 627.321,A -85,B 0,C 180,E1 -1426.154,E2 -1426.154} C_VEL
LIN {X 0,Y 587.344,Z 627.316,A -85,B 0,C 180,E1 -1428.963,E2 -1428.963} C_VEL
LIN {X 0,Y 587.374,Z 627.32,A -85,B 0,C 180,E1 -1431.745,E2 -1431.745} C_VEL
LIN {X 0,Y 587.354,Z 627.318,A -85,B 0,C 180,E1 -1434.507,E2 -1434.507} C_VEL
LIN {X 0,Y 587.379,Z 627.312,A -85,B 0,C 180,E1 -1437.257,E2 -1437.257} C_VEL
LIN {X 0,Y 587.386,Z 627.321,A -85,B 0,C 180,E1 -1440,E2 -1440} C_VEL
LIN {X 0,Y 587.379,Z 627.314,A -85,B 0,C 180,E1 -1442.743,E2 -1442.743} C_VEL
LIN {X 0,Y 587.354,Z 627.316,A -85,B 0,C 180,E1 -1445.493,E2 -1445.493} C_VEL
LIN {X 0,Y 587.374,Z 627.322,A -85,B 0,C 180,E1 -1448.255,E2 -1448.255} C_VEL
LIN {X 0,Y 587.349,Z 627.316,A -85,B 0,C 180,E1 -1451.134,E2 -1451.134} C_VEL
LIN {X 0,Y 587.366,Z 627.324,A -85,B 0,C 180,E1 -1454.261,E2 -1454.261} C_VEL
LIN {X 0,Y 587.351,Z 627.315,A -85,B 0,C 180,E1 -1457.406,E2 -1457.406} C_VEL
LIN {X 0,Y 587.332,Z 627.328,A -85,B 0,C 180,E1 -1460.305,E2 -1460.305} C_VEL
LIN {X 0,Y 587.324,Z 627.319,A -85,B 0,C 180,E1 -1463.259,E2 -1463.259} C_VEL
LIN {X 0,Y 587.335,Z 627.317,A -85,B 0,C 180,E1 -1465.517,E2 -1465.517} C_VEL
LIN {X 0,Y 587.349,Z 627.317,A -85,B 0,C 180,E1 -1467.818,E2 -1467.818} C_VEL
LIN {X 0,Y 587.339,Z 627.328,A -85,B 0,C 180,E1 -1470.51,E2 -1470.51} C_VEL
LIN {X 0,Y 587.335,Z 627.318,A -85,B 0,C 180,E1 -1473.397,E2 -1473.397} C_VEL
LIN {X 0,Y 587.293,Z 627.324,A -85,B 0,C 180,E1 -1475.9,E2 -1475.9} C_VEL
LIN {X 0,Y 587.333,Z 627.327,A -85,B 0,C 180,E1 -1478.479,E2 -1478.479} C_VEL
LIN {X 0,Y 587.338,Z 627.32,A -85,B 0,C 180,E1 -1481.157,E2 -1481.157} C_VEL
LIN {X 0,Y 587.337,Z 627.32,A -85,B 0,C 180,E1 -1484.114,E2 -1484.114} C_VEL
LIN {X 0,Y 587.316,Z 627.328,A -85,B 0,C 180,E1 -1486.994,E2 -1486.994} C_VEL
LIN {X 0,Y 587.319,Z 627.322,A -85,B 0,C 180,E1 -1489.746,E2 -1489.746} C_VEL
LIN {X 0,Y 587.346,Z 627.323,A -85,B 0,C 180,E1 -1492.392,E2 -1492.392} C_VEL
LIN {X 0,Y 587.342,Z 627.441,A -85,B 0,C 180,E1 -1493.599,E2 -1493.599} C_VEL
LIN {X 0,Y 587.937,Z 631.219,A -85,B 0,C 180,E1 -1494.376,E2 -1494.376} C_VEL
LIN {X 0,Y 588.053,Z 645.495,A -85,B 0,C 180,E1 -1497.128,E2 -1497.128} C_VEL
LIN {X 0,Y 588.009,Z 656.74,A -85,B 0,C 180,E1 -1499.38,E2 -1499.38} C_VEL
LIN {X 0,Y 587.853,Z 670.919,A -85,B 0,C 180,E1 -1502.215,E2 -1502.215} C_VEL
LIN {X 0,Y 587.716,Z 684.58,A -85,B 0,C 180,E1 -1504.88,E2 -1504.88} C_VEL
LIN {X 0,Y 587.611,Z 698.275,A -85,B 0,C 180,E1 -1507.497,E2 -1507.497} C_VEL
LIN {X 0,Y 587.52,Z 713.926,A -85,B 0,C 180,E1 -1510.431,E2 -1510.431} C_VEL
LIN {X 0,Y 587.425,Z 729.578,A -85,B 0,C 180,E1 -1513.313,E2 -1513.313} C_VEL
LIN {X 0,Y 587.345,Z 745.229,A -85,B 0,C 180,E1 -1516.154,E2 -1516.154} C_VEL
LIN {X 0,Y 587.313,Z 754.155,A -85,B 0,C 180,E1 -1517.758,E2 -1517.758} C_VEL
LIN {X 0,Y 587.742,Z 759.932,A -85,B 0,C 180,E1 -1517.855,E2 -1517.855} C_VEL
LIN {X 0,Y 587.681,Z 773.205,A -85,B 0,C 180,E1 -1518.16,E2 -1518.16} C_VEL
LIN {X 0,Y 587.623,Z 785.729,A -85,B 0,C 180,E1 -1518.589,E2 -1518.589} C_VEL
LIN {X 0,Y 587.522,Z 797.628,A -85,B 0,C 180,E1 -1519.14,E2 -1519.14} C_VEL
LIN {X 0,Y 587.461,Z 809.196,A -85,B 0,C 180,E1 -1519.836,E2 -1519.836} C_VEL
LIN {X 0,Y 587.367,Z 819.592,A -85,B 0,C 180,E1 -1520.617,E2 -1520.617} C_VEL
LIN {X 0,Y 587.322,Z 828.109,A -85,B 0,C 180,E1 -1521.397,E2 -1521.397} C_VEL
LIN {X 0,Y 587.274,Z 835.958,A -85,B 0,C 180,E1 -1522.262,E2 -1522.262} C_VEL
LIN {X 0,Y 587.231,Z 842.468,A -85,B 0,C 180,E1 -1523.126,E2 -1523.126} C_VEL
LIN {X 0,Y 587.236,Z 848.865,A -85,B 0,C 180,E1 -1524.161,E2 -1524.161} C_VEL
LIN {X 0,Y 587.147,Z 853.948,A -85,B 0,C 180,E1 -1525.193,E2 -1525.193} C_VEL
LIN {X 0,Y 587.213,Z 857.895,A -85,B 0,C 180,E1 -1526.225,E2 -1526.225} C_VEL
LIN {X 0,Y 587.132,Z 860.809,A -85,B 0,C 180,E1 -1527.255,E2 -1527.255} C_VEL
LIN {X 0,Y 587.138,Z 862.201,A -85,B 0,C 180,E1 -1527.942,E2 -1527.942} C_VEL
LIN {X 0,Y 587.14,Z 863.784,A -85,B 0,C 180,E1 -1529.314,E2 -1529.314} C_VEL
LIN {X 0,Y 587.137,Z 864,A -85,B 0,C 180,E1 -1530,E2 -1530} C_VEL
LIN {X 0,Y 587.147,Z 863.185,A -85,B 0,C 180,E1 -1531.371,E2 -1531.371} C_VEL
LIN {X 0,Y 587.138,Z 862.202,A -85,B 0,C 180,E1 -1532.058,E2 -1532.058} C_VEL
LIN {X 0,Y 587.132,Z 860.81,A -85,B 0,C 180,E1 -1532.744,E2 -1532.744} C_VEL
LIN {X 0,Y 587.213,Z 857.897,A -85,B 0,C 180,E1 -1533.774,E2 -1533.774} C_VEL
LIN {X 0,Y 587.147,Z 853.952,A -85,B 0,C 180,E1 -1534.806,E2 -1534.806} C_VEL
LIN {X 0,Y 587.217,Z 847.88,A -85,B 0,C 180,E1 -1536.011,E2 -1536.011} C_VEL
LIN {X 0,Y 587.245,Z 841.239,A -85,B 0,C 180,E1 -1537.046,E2 -1537.046} C_VEL
LIN {X 0,Y 587.299,Z 832.993,A -85,B 0,C 180,E1 -1538.083,E2 -1538.083} C_VEL
LIN {X 0,Y 587.343,Z 824.542,A -85,B 0,C 180,E1 -1538.949,E2 -1538.949} C_VEL
LIN {X 0,Y 587.415,Z 814.1,A -85,B 0,C 180,E1 -1539.816,E2 -1539.816} C_VEL
LIN {X 0,Y 587.5,Z 803.766,A -85,B 0,C 180,E1 -1540.511,E2 -1540.511} C_VEL
LIN {X 0,Y 587.562,Z 792.05,A -85,B 0,C 180,E1 -1541.138,E2 -1541.138} C_VEL
LIN {X 0,Y 587.629,Z 779.645,A -85,B 0,C 180,E1 -1541.638,E2 -1541.638} C_VEL
LIN {X 0,Y 587.709,Z 766.459,A -85,B 0,C 180,E1 -1542.013,E2 -1542.013} C_VEL
LIN {X 0,Y 587.517,Z 755.633,A -85,B 0,C 180,E1 -1542.215,E2 -1542.215} C_VEL
LIN {X 0,Y 587.317,Z 754.037,A -85,B 0,C 180,E1 -1542.263,E2 -1542.263} C_VEL
LIN {X 0,Y 587.381,Z 737.407,A -85,B 0,C 180,E1 -1545.261,E2 -1545.261} C_VEL
LIN {X 0,Y 587.466,Z 721.756,A -85,B 0,C 180,E1 -1548.122,E2 -1548.122} C_VEL
LIN {X 0,Y 587.558,Z 708.061,A -85,B 0,C 180,E1 -1550.662,E2 -1550.662} C_VEL
LIN {X 0,Y 587.648,Z 692.41,A -85,B 0,C 180,E1 -1553.618,E2 -1553.618} C_VEL
LIN {X 0,Y 587.787,Z 678.671,A -85,B 0,C 180,E1 -1556.265,E2 -1556.265} C_VEL
LIN {X 0,Y 587.905,Z 665.302,A -85,B 0,C 180,E1 -1558.9,E2 -1558.9} C_VEL
LIN {X 0,Y 588.044,Z 651.326,A -85,B 0,C 180,E1 -1561.726,E2 -1561.726} C_VEL
LIN {X 0,Y 588.028,Z 638.783,A -85,B 0,C 180,E1 -1564.175,E2 -1564.175} C_VEL
LIN {X 0,Y 587.954,Z 630.484,A -85,B 0,C 180,E1 -1565.853,E2 -1565.853} C_VEL
LIN {X 0,Y 587.345,Z 627.324,A -85,B 0,C 180,E1 -1566.576,E2 -1566.576} C_VEL
LIN {X 0,Y 587.346,Z 627.322,A -85,B 0,C 180,E1 -1569.358,E2 -1569.358} C_VEL
LIN {X 0,Y 587.333,Z 627.321,A -85,B 0,C 180,E1 -1572.107,E2 -1572.107} C_VEL
LIN {X 0,Y 587.314,Z 627.325,A -85,B 0,C 180,E1 -1575.088,E2 -1575.088} C_VEL
LIN {X 0,Y 587.35,Z 627.319,A -85,B 0,C 180,E1 -1577.927,E2 -1577.927} C_VEL
LIN {X 0,Y 587.334,Z 627.32,A -85,B 0,C 180,E1 -1581.057,E2 -1581.057} C_VEL
LIN {X 0,Y 587.351,Z 627.317,A -85,B 0,C 180,E1 -1583.291,E2 -1583.291} C_VEL
LIN {X 0,Y 587.357,Z 627.321,A -85,B 0,C 180,E1 -1585.779,E2 -1585.779} C_VEL
LIN {X 0,Y 587.347,Z 627.322,A -85,B 0,C 180,E1 -1588.231,E2 -1588.231} C_VEL
LIN {X 0,Y 587.346,Z 627.317,A -85,B 0,C 180,E1 -1590.866,E2 -1590.866} C_VEL
LIN {X 0,Y 587.357,Z 627.323,A -85,B 0,C 180,E1 -1593.818,E2 -1593.818} C_VEL
LIN {X 0,Y 587.335,Z 627.322,A -85,B 0,C 180,E1 -1595.993,E2 -1595.993} C_VEL
LIN {X 0,Y 587.344,Z 627.322,A -85,B 0,C 180,E1 -1598.963,E2 -1598.963} C_VEL
LIN {X 0,Y 587.324,Z 627.321,A -85,B 0,C 180,E1 -1601.873,E2 -1601.873} C_VEL
LIN {X 0,Y 587.322,Z 627.321,A -85,B 0,C 180,E1 -1604.025,E2 -1604.025} C_VEL
LIN {X 0,Y 587.357,Z 627.317,A -85,B 0,C 180,E1 -1606.154,E2 -1606.154} C_VEL
LIN {X 0,Y 587.341,Z 627.326,A -85,B 0,C 180,E1 -1608.962,E2 -1608.962} C_VEL
LIN {X 0,Y 587.368,Z 627.315,A -85,B 0,C 180,E1 -1611.745,E2 -1611.745} C_VEL
LIN {X 0,Y 587.351,Z 627.326,A -85,B 0,C 180,E1 -1614.507,E2 -1614.507} C_VEL
LIN {X 0,Y 587.376,Z 627.314,A -85,B 0,C 180,E1 -1617.257,E2 -1617.257} C_VEL
LIN {X 0,Y 587.378,Z 627.32,A -85,B 0,C 180,E1 -1620,E2 -1620} C_VEL
LIN {X 0,Y 587.377,Z 627.316,A -85,B 0,C 180,E1 -1622.743,E2 -1622.743} C_VEL
LIN {X 0,Y 587.403,Z 627.484,A -85,B 0,C 180,E1 -1625.32,E2 -1625.32} C_VEL
LIN {X 0,Y 587.631,Z 637.308,A -85,B 0,C 180,E1 -1627.56,E2 -1627.56} C_VEL
LIN {X 0,Y 587.779,Z 646.221,A -85,B 0,C 180,E1 -1629.636,E2 -1629.636} C_VEL
LIN {X 0,Y 587.645,Z 658.475,A -85,B 0,C 180,E1 -1632.783,E2 -1632.783} C_VEL
LIN {X 0,Y 587.544,Z 669.805,A -85,B 0,C 180,E1 -1635.613,E2 -1635.613} C_VEL
LIN {X 0,Y 587.501,Z 676.92,A -85,B 0,C 180,E1 -1637.358,E2 -1637.358} C_VEL
LIN {X 0,Y 586.869,Z 679.197,A -85,B 0,C 180,E1 -1637.886,E2 -1637.886} C_VEL
LIN {X 0,Y 583.997,Z 683.158,A -85,B 0,C 180,E1 -1638.73,E2 -1638.73} C_VEL
LIN {X 0,Y 581.092,Z 687.141,A -85,B 0,C 180,E1 -1639.582,E2 -1639.582} C_VEL
LIN {X 0,Y 580.427,Z 689.456,A -85,B 0,C 180,E1 -1640.117,E2 -1640.117} C_VEL
LIN {X 0,Y 580.318,Z 701.563,A -85,B 0,C 180,E1 -1643.017,E2 -1643.017} C_VEL
LIN {X 0,Y 580.242,Z 713.586,A -85,B 0,C 180,E1 -1645.851,E2 -1645.851} C_VEL
LIN {X 0,Y 580.195,Z 725.546,A -85,B 0,C 180,E1 -1648.635,E2 -1648.635} C_VEL
LIN {X 0,Y 580.236,Z 726.191,A -85,B 0,C 180,E1 -1648.682,E2 -1648.682} C_VEL
LIN {X 0,Y 580.805,Z 731.114,A -85,B 0,C 180,E1 -1648.775,E2 -1648.775} C_VEL
LIN {X 0,Y 580.735,Z 744.659,A -85,B 0,C 180,E1 -1649.103,E2 -1649.103} C_VEL
LIN {X 0,Y 580.634,Z 757.424,A -85,B 0,C 180,E1 -1649.565,E2 -1649.565} C_VEL
LIN {X 0,Y 580.518,Z 769.556,A -85,B 0,C 180,E1 -1650.16,E2 -1650.16} C_VEL
LIN {X 0,Y 580.438,Z 781.457,A -85,B 0,C 180,E1 -1650.914,E2 -1650.914} C_VEL
LIN {X 0,Y 580.35,Z 791.222,A -85,B 0,C 180,E1 -1651.686,E2 -1651.686} C_VEL
LIN {X 0,Y 580.265,Z 800.731,A -85,B 0,C 180,E1 -1652.614,E2 -1652.614} C_VEL
LIN {X 0,Y 580.2,Z 808.626,A -85,B 0,C 180,E1 -1653.554,E2 -1653.554} C_VEL
LIN {X 0,Y 580.166,Z 816.4,A -85,B 0,C 180,E1 -1654.705,E2 -1654.705} C_VEL
LIN {X 0,Y 580.097,Z 821.931,A -85,B 0,C 180,E1 -1655.737,E2 -1655.737} C_VEL
LIN {X 0,Y 580.084,Z 826.789,A -85,B 0,C 180,E1 -1656.907,E2 -1656.907} C_VEL
LIN {X 0,Y 580.065,Z 830.547,A -85,B 0,C 180,E1 -1658.164,E2 -1658.164} C_VEL
LIN {X 0,Y 580.042,Z 832.507,A -85,B 0,C 180,E1 -1659.156,E2 -1659.156} C_VEL
LIN {X 0,Y 580.035,Z 833.711,A -85,B 0,C 180,E1 -1660.242,E2 -1660.242} C_VEL
LIN {X 0,Y 580.032,Z 833.948,A -85,B 0,C 180,E1 -1661.304,E2 -1661.304} C_VEL
LIN {X 0,Y 580.053,Z 832.836,A -85,B 0,C 180,E1 -1662.727,E2 -1662.727} C_VEL
LIN {X 0,Y 580.034,Z 831.116,A -85,B 0,C 180,E1 -1663.681,E2 -1663.681} C_VEL
LIN {X 0,Y 580.078,Z 828.573,A -85,B 0,C 180,E1 -1664.644,E2 -1664.644} C_VEL
LIN {X 0,Y 580.099,Z 825.11,A -85,B 0,C 180,E1 -1665.626,E2 -1665.626} C_VEL
LIN {X 0,Y 580.121,Z 820.587,A -85,B 0,C 180,E1 -1666.626,E2 -1666.626} C_VEL
LIN {X 0,Y 580.137,Z 814.805,A -85,B 0,C 180,E1 -1667.644,E2 -1667.644} C_VEL
LIN {X 0,Y 580.195,Z 807.523,A -85,B 0,C 180,E1 -1668.678,E2 -1668.678} C_VEL
LIN {X 0,Y 580.268,Z 798.31,A -85,B 0,C 180,E1 -1669.732,E2 -1669.732} C_VEL
LIN {X 0,Y 580.386,Z 788.045,A -85,B 0,C 180,E1 -1670.67,E2 -1670.67} C_VEL
LIN {X 0,Y 580.461,Z 777.856,A -85,B 0,C 180,E1 -1671.426,E2 -1671.426} C_VEL
LIN {X 0,Y 580.554,Z 766.511,A -85,B 0,C 180,E1 -1672.095,E2 -1672.095} C_VEL
LIN {X 0,Y 580.651,Z 754.346,A -85,B 0,C 180,E1 -1672.65,E2 -1672.65} C_VEL
LIN {X 0,Y 580.762,Z 741.247,A -85,B 0,C 180,E1 -1673.085,E2 -1673.085} C_VEL
LIN {X 0,Y 580.695,Z 728.977,A -85,B 0,C 180,E1 -1673.356,E2 -1673.356} C_VEL
LIN {X 0,Y 580.18,Z 725.635,A -85,B 0,C 180,E1 -1673.435,E2 -1673.435} C_VEL
LIN {X 0,Y 580.232,Z 714.007,A -85,B 0,C 180,E1 -1676.14,E2 -1676.14} C_VEL
LIN {X 0,Y 580.313,Z 701.909,A -85,B 0,C 180,E1 -1678.991,E2 -1678.991} C_VEL
LIN {X 0,Y 580.394,Z 690.091,A -85,B 0,C 180,E1 -1681.82,E2 -1681.82} C_VEL
LIN {X 0,Y 580.492,Z 678.905,A -85,B 0,C 180,E1 -1684.546,E2 -1684.546} C_VEL
LIN {X 0,Y 580.576,Z 668.192,A -85,B 0,C 180,E1 -1687.21,E2 -1687.21} C_VEL
LIN {X 0,Y 580.693,Z 657.907,A -85,B 0,C 180,E1 -1689.823,E2 -1689.823} C_VEL
LIN {X 0,Y 580.762,Z 647.805,A -85,B 0,C 180,E1 -1692.391,E2 -1692.391} C_VEL
LIN {X 0,Y 580.716,Z 637.437,A -85,B 0,C 180,E1 -1694.919,E2 -1694.919} C_VEL
LIN {X 0,Y 580.566,Z 630.06,A -85,B 0,C 180,E1 -1696.703,E2 -1696.703} C_VEL
LIN {X 0,Y 580.321,Z 628.202,A -85,B 0,C 180,E1 -1697.187,E2 -1697.187} C_VEL
LIN {X 0,Y 580.302,Z 628.201,A -85,B 0,C 180,E1 -1699.534,E2 -1699.534} C_VEL
LIN {X 0,Y 580.331,Z 628.197,A -85,B 0,C 180,E1 -1702.345,E2 -1702.345} C_VEL
LIN {X 0,Y 580.34,Z 628.197,A -85,B 0,C 180,E1 -1705.138,E2 -1705.138} C_VEL
LIN {X 0,Y 580.344,Z 628.198,A -85,B 0,C 180,E1 -1707.918,E2 -1707.918} C_VEL
LIN {X 0,Y 580.369,Z 628.196,A -85,B 0,C 180,E1 -1710.694,E2 -1710.694} C_VEL
LIN {X 0,Y 580.29,Z 628.205,A -85,B 0,C 180,E1 -1713.472,E2 -1713.472} C_VEL
LIN {X 0,Y 580.322,Z 628.198,A -85,B 0,C 180,E1 -1715.56,E2 -1715.56} C_VEL
LIN {X 0,Y 580.338,Z 628.197,A -85,B 0,C 180,E1 -1718.356,E2 -1718.356} C_VEL
LIN {X 0,Y 580.303,Z 628.202,A -85,B 0,C 180,E1 -1721.191,E2 -1721.191} C_VEL
LIN {X 0,Y 580.33,Z 628.201,A -85,B 0,C 180,E1 -1724.017,E2 -1724.017} C_VEL
LIN {X 0,Y 580.317,Z 628.2,A -85,B 0,C 180,E1 -1726.915,E2 -1726.915} C_VEL
LIN {X 0,Y 580.29,Z 628.202,A -85,B 0,C 180,E1 -1729.823,E2 -1729.823} C_VEL
LIN {X 0,Y 580.277,Z 628.207,A -85,B 0,C 180,E1 -1732.053,E2 -1732.053} C_VEL
LIN {X 0,Y 580.309,Z 628.2,A -85,B 0,C 180,E1 -1735.08,E2 -1735.08} C_VEL
LIN {X 0,Y 580.327,Z 628.252,A -85,B 0,C 180,E1 -1736.214,E2 -1736.214} C_VEL
LIN {X 0,Y 580.653,Z 633.483,A -85,B 0,C 180,E1 -1736.406,E2 -1736.406} C_VEL
LIN {X 0,Y 580.592,Z 644.614,A -85,B 0,C 180,E1 -1736.899,E2 -1736.899} C_VEL
LIN {X 0,Y 580.489,Z 655.932,A -85,B 0,C 180,E1 -1737.544,E2 -1737.544} C_VEL
LIN {X 0,Y 580.416,Z 664.983,A -85,B 0,C 180,E1 -1738.18,E2 -1738.18} C_VEL
LIN {X 0,Y 580.31,Z 674.352,A -85,B 0,C 180,E1 -1738.975,E2 -1738.975} C_VEL
LIN {X 0,Y 580.23,Z 682.179,A -85,B 0,C 180,E1 -1739.776,E2 -1739.776} C_VEL
LIN {X 0,Y 580.197,Z 690.538,A -85,B 0,C 180,E1 -1740.813,E2 -1740.813} C_VEL
LIN {X 0,Y 580.153,Z 698.158,A -85,B 0,C 180,E1 -1742.007,E2 -1742.007} C_VEL
LIN {X 0,Y 580.091,Z 703.323,A -85,B 0,C 180,E1 -1743.038,E2 -1743.038} C_VEL
LIN {X 0,Y 580.08,Z 707.774,A -85,B 0,C 180,E1 -1744.197,E2 -1744.197} C_VEL
LIN {X 0,Y 580.042,Z 710.483,A -85,B 0,C 180,E1 -1745.137,E2 -1745.137} C_VEL
LIN {X 0,Y 580.015,Z 712.88,A -85,B 0,C 180,E1 -1746.422,E2 -1746.422} C_VEL
LIN {X 0,Y 580.027,Z 713.744,A -85,B 0,C 180,E1 -1747.289,E2 -1747.289} C_VEL
LIN {X 0,Y 580.016,Z 713.979,A -85,B 0,C 180,E1 -1748.168,E2 -1748.168} C_VEL
LIN {X 0,Y 580.019,Z 713.497,A -85,B 0,C 180,E1 -1749.152,E2 -1749.152} C_VEL
LIN {X 0,Y 580.044,Z 712.014,A -85,B 0,C 180,E1 -1750.242,E2 -1750.242} C_VEL
LIN {X 0,Y 580.043,Z 709.587,A -85,B 0,C 180,E1 -1751.304,E2 -1751.304} C_VEL
LIN {X 0,Y 580.092,Z 706.197,A -85,B 0,C 180,E1 -1752.351,E2 -1752.351} C_VEL
LIN {X 0,Y 580.109,Z 701.844,A -85,B 0,C 180,E1 -1753.373,E2 -1753.373} C_VEL
LIN {X 0,Y 580.155,Z 696.438,A -85,B 0,C 180,E1 -1754.379,E2 -1754.379} C_VEL
LIN {X 0,Y 580.17,Z 689.891,A -85,B 0,C 180,E1 -1755.365,E2 -1755.365} C_VEL
LIN {X 0,Y 580.228,Z 681.967,A -85,B 0,C 180,E1 -1756.337,E2 -1756.337} C_VEL
LIN {X 0,Y 580.311,Z 673.665,A -85,B 0,C 180,E1 -1757.179,E2 -1757.179} C_VEL
LIN {X 0,Y 580.437,Z 663.635,A -85,B 0,C 180,E1 -1758.014,E2 -1758.014} C_VEL
LIN {X 0,Y 580.486,Z 652.4,A -85,B 0,C 180,E1 -1758.769,E2 -1758.769} C_VEL
LIN {X 0,Y 580.62,Z 639.779,A -85,B 0,C 180,E1 -1759.419,E2 -1759.419} C_VEL
LIN {X 0,Y 580.682,Z 629.872,A -85,B 0,C 180,E1 -1759.814,E2 -1759.814} C_VEL
LIN {X 0,Y 580.316,Z 628.198,A -85,B 0,C 180,E1 -1759.891,E2 -1759.891} C_VEL
LIN {X 0,Y 580.3,Z 628.198,A -85,B 0,C 180,E1 -1763.066,E2 -1763.066} C_VEL
LIN {X 0,Y 580.318,Z 628.195,A -85,B 0,C 180,E1 -1766.145,E2 -1766.145} C_VEL
LIN {X 0,Y 580.278,Z 628.197,A -85,B 0,C 180,E1 -1768.615,E2 -1768.615} C_VEL
LIN {X 0,Y 580.294,Z 628.196,A -85,B 0,C 180,E1 -1771.024,E2 -1771.024} C_VEL
LIN {X 0,Y 580.293,Z 628.205,A -85,B 0,C 180,E1 -1773.666,E2 -1773.666} C_VEL
LIN {X 0,Y 580.301,Z 628.204,A -85,B 0,C 180,E1 -1775.684,E2 -1775.684} C_VEL
LIN {X 0,Y 580.273,Z 628.205,A -85,B 0,C 180,E1 -1777.947,E2 -1777.947} C_VEL
LIN {X 0,Y 580.301,Z 628.194,A -85,B 0,C 180,E1 -1780.914,E2 -1780.914} C_VEL
LIN {X 0,Y 580.281,Z 628.207,A -85,B 0,C 180,E1 -1783.826,E2 -1783.826} C_VEL
LIN {X 0,Y 580.326,Z 628.2,A -85,B 0,C 180,E1 -1785.983,E2 -1785.983} C_VEL
LIN {X 0,Y 580.306,Z 628.193,A -85,B 0,C 180,E1 -1788.827,E2 -1788.827} C_VEL
LIN {X 0,Y 580.336,Z 628.195,A -85,B 0,C 180,E1 -1791.644,E2 -1791.644} C_VEL
LIN {X 0,Y 580.321,Z 628.195,A -85,B 0,C 180,E1 -1794.44,E2 -1794.44} C_VEL
LIN {X 0,Y 580.344,Z 628.188,A -85,B 0,C 180,E1 -1797.224,E2 -1797.224} C_VEL
LIN {X 0,Y 580.355,Z 628.197,A -85,B 0,C 180,E1 -1800,E2 -1800} C_VEL
LIN {X 0,Y 580.344,Z 628.19,A -85,B 0,C 180,E1 -1802.777,E2 -1802.777} C_VEL
LIN {X 0,Y 580.322,Z 628.192,A -85,B 0,C 180,E1 -1805.56,E2 -1805.56} C_VEL
LIN {X 0,Y 580.337,Z 628.196,A -85,B 0,C 180,E1 -1808.356,E2 -1808.356} C_VEL
LIN {X 0,Y 580.301,Z 628.194,A -85,B 0,C 180,E1 -1811.191,E2 -1811.191} C_VEL
LIN {X 0,Y 580.327,Z 628.196,A -85,B 0,C 180,E1 -1814.017,E2 -1814.017} C_VEL
LIN {X 0,Y 580.314,Z 628.194,A -85,B 0,C 180,E1 -1816.914,E2 -1816.914} C_VEL
LIN {X 0,Y 580.29,Z 628.197,A -85,B 0,C 180,E1 -1819.823,E2 -1819.823} C_VEL
LIN {X 0,Y 580.274,Z 628.202,A -85,B 0,C 180,E1 -1822.053,E2 -1822.053} C_VEL
LIN {X 0,Y 580.308,Z 628.194,A -85,B 0,C 180,E1 -1825.08,E2 -1825.08} C_VEL
LIN {X 0,Y 580.302,Z 628.2,A -85,B 0,C 180,E1 -1828.186,E2 -1828.186} C_VEL
LIN {X 0,Y 580.286,Z 628.203,A -85,B 0,C 180,E1 -1830.695,E2 -1830.695} C_VEL
LIN {X 0,Y 580.305,Z 628.194,A -85,B 0,C 180,E1 -1833.316,E2 -1833.316} C_VEL
LIN {X 0,Y 580.247,Z 628.202,A -85,B 0,C 180,E1 -1835.756,E2 -1835.756} C_VEL
LIN {X 0,Y 580.291,Z 628.199,A -85,B 0,C 180,E1 -1838.146,E2 -1838.146} C_VEL
LIN {X 0,Y 580.302,Z 628.202,A -85,B 0,C 180,E1 -1840.843,E2 -1840.843} C_VEL
LIN {X 0,Y 580.291,Z 628.195,A -85,B 0,C 180,E1 -1843.657,E2 -1843.657} C_VEL
LIN {X 0,Y 580.277,Z 628.207,A -85,B 0,C 180,E1 -1846.61,E2 -1846.61} C_VEL
LIN {X 0,Y 580.301,Z 628.201,A -85,B 0,C 180,E1 -1849.157,E2 -1849.157} C_VEL
LIN {X 0,Y 580.29,Z 628.199,A -85,B 0,C 180,E1 -1851.927,E2 -1851.927} C_VEL
LIN {X 0,Y 580.336,Z 628.375,A -85,B 0,C 180,E1 -1853.411,E2 -1853.411} C_VEL
LIN {X 0,Y 581.04,Z 633.644,A -85,B 0,C 180,E1 -1854.508,E2 -1854.508} C_VEL
LIN {X 0,Y 581.123,Z 647.641,A -85,B 0,C 180,E1 -1857.235,E2 -1857.235} C_VEL
LIN {X 0,Y 581.142,Z 659.147,A -85,B 0,C 180,E1 -1859.474,E2 -1859.474} C_VEL
LIN {X 0,Y 580.932,Z 673.273,A -85,B 0,C 180,E1 -1862.326,E2 -1862.326} C_VEL
LIN {X 0,Y 580.768,Z 687.733,A -85,B 0,C 180,E1 -1865.175,E2 -1865.175} C_VEL
LIN {X 0,Y 580.622,Z 702.188,A -85,B 0,C 180,E1 -1867.961,E2 -1867.961} C_VEL
LIN {X 0,Y 580.493,Z 717.173,A -85,B 0,C 180,E1 -1870.795,E2 -1870.795} C_VEL
LIN {X 0,Y 580.394,Z 731.534,A -85,B 0,C 180,E1 -1873.467,E2 -1873.467} C_VEL
LIN {X 0,Y 580.297,Z 747.185,A -85,B 0,C 180,E1 -1876.339,E2 -1876.339} C_VEL
LIN {X 0,Y 580.253,Z 754.155,A -85,B 0,C 180,E1 -1877.607,E2 -1877.607} C_VEL
LIN {X 0,Y 580.824,Z 759.931,A -85,B 0,C 180,E1 -1877.708,E2 -1877.708} C_VEL
LIN {X 0,Y 580.75,Z 773.205,A -85,B 0,C 180,E1 -1878.017,E2 -1878.017} C_VEL
LIN {X 0,Y 580.674,Z 785.361,A -85,B 0,C 180,E1 -1878.436,E2 -1878.436} C_VEL
LIN {X 0,Y 580.544,Z 797.627,A -85,B 0,C 180,E1 -1879.008,E2 -1879.008} C_VEL
LIN {X 0,Y 580.43,Z 809.197,A -85,B 0,C 180,E1 -1879.712,E2 -1879.712} C_VEL
LIN {X 0,Y 580.346,Z 819.593,A -85,B 0,C 180,E1 -1880.503,E2 -1880.503} C_VEL
LIN {X 0,Y 580.272,Z 828.109,A -85,B 0,C 180,E1 -1881.292,E2 -1881.292} C_VEL
LIN {X 0,Y 580.222,Z 835.958,A -85,B 0,C 180,E1 -1882.168,E2 -1882.168} C_VEL
LIN {X 0,Y 580.154,Z 843.649,A -85,B 0,C 180,E1 -1883.221,E2 -1883.221} C_VEL
LIN {X 0,Y 580.139,Z 850.678,A -85,B 0,C 180,E1 -1884.438,E2 -1884.438} C_VEL
LIN {X 0,Y 580.108,Z 855.37,A -85,B 0,C 180,E1 -1885.483,E2 -1885.483} C_VEL
LIN {X 0,Y 580.123,Z 858.956,A -85,B 0,C 180,E1 -1886.527,E2 -1886.527} C_VEL
LIN {X 0,Y 580.043,Z 860.809,A -85,B 0,C 180,E1 -1887.222,E2 -1887.222} C_VEL
LIN {X 0,Y 580.038,Z 862.201,A -85,B 0,C 180,E1 -1887.917,E2 -1887.917} C_VEL
LIN {X 0,Y 580.04,Z 863.784,A -85,B 0,C 180,E1 -1889.305,E2 -1889.305} C_VEL
LIN {X 0,Y 580.037,Z 864,A -85,B 0,C 180,E1 -1890,E2 -1890} C_VEL
LIN {X 0,Y 580.047,Z 863.185,A -85,B 0,C 180,E1 -1891.388,E2 -1891.388} C_VEL
LIN {X 0,Y 580.038,Z 862.201,A -85,B 0,C 180,E1 -1892.083,E2 -1892.083} C_VEL
LIN {X 0,Y 580.043,Z 860.81,A -85,B 0,C 180,E1 -1892.778,E2 -1892.778} C_VEL
LIN {X 0,Y 580.11,Z 857.897,A -85,B 0,C 180,E1 -1893.82,E2 -1893.82} C_VEL
LIN {X 0,Y 580.054,Z 853.952,A -85,B 0,C 180,E1 -1894.865,E2 -1894.865} C_VEL
LIN {X 0,Y 580.139,Z 847.88,A -85,B 0,C 180,E1 -1896.084,E2 -1896.084} C_VEL
LIN {X 0,Y 580.184,Z 841.24,A -85,B 0,C 180,E1 -1897.132,E2 -1897.132} C_VEL
LIN {X 0,Y 580.25,Z 832.994,A -85,B 0,C 180,E1 -1898.181,E2 -1898.181} C_VEL
LIN {X 0,Y 580.308,Z 824.542,A -85,B 0,C 180,E1 -1899.058,E2 -1899.058} C_VEL
LIN {X 0,Y 580.414,Z 814.101,A -85,B 0,C 180,E1 -1899.936,E2 -1899.936} C_VEL
LIN {X 0,Y 580.52,Z 803.765,A -85,B 0,C 180,E1 -1900.639,E2 -1900.639} C_VEL
LIN {X 0,Y 580.571,Z 792.602,A -85,B 0,C 180,E1 -1901.247,E2 -1901.247} C_VEL
LIN {X 0,Y 580.68,Z 780.784,A -85,B 0,C 180,E1 -1901.74,E2 -1901.74} C_VEL
LIN {X 0,Y 580.784,Z 767.373,A -85,B 0,C 180,E1 -1902.137,E2 -1902.137} C_VEL
LIN {X 0,Y 580.631,Z 756.576,A -85,B 0,C 180,E1 -1902.348,E2 -1902.348} C_VEL
LIN {X 0,Y 580.252,Z 754.037,A -85,B 0,C 180,E1 -1902.414,E2 -1902.414} C_VEL
LIN {X 0,Y 580.341,Z 739.364,A -85,B 0,C 180,E1 -1905.091,E2 -1905.091} C_VEL
LIN {X 0,Y 580.441,Z 723.713,A -85,B 0,C 180,E1 -1907.984,E2 -1907.984} C_VEL
LIN {X 0,Y 580.585,Z 708.204,A -85,B 0,C 180,E1 -1910.895,E2 -1910.895} C_VEL
LIN {X 0,Y 580.734,Z 692.41,A -85,B 0,C 180,E1 -1913.916,E2 -1913.916} C_VEL
LIN {X 0,Y 580.882,Z 678.715,A -85,B 0,C 180,E1 -1916.593,E2 -1916.593} C_VEL
LIN {X 0,Y 581.057,Z 664.474,A -85,B 0,C 180,E1 -1919.442,E2 -1919.442} C_VEL
LIN {X 0,Y 581.127,Z 653.021,A -85,B 0,C 180,E1 -1921.74,E2 -1921.74} C_VEL
LIN {X 0,Y 581.115,Z 640.32,A -85,B 0,C 180,E1 -1924.219,E2 -1924.219} C_VEL
LIN {X 0,Y 581.087,Z 632.314,A -85,B 0,C 180,E1 -1925.871,E2 -1925.871} C_VEL
LIN {X 0,Y 580.304,Z 628.201,A -85,B 0,C 180,E1 -1926.782,E2 -1926.782} C_VEL
LIN {X 0,Y 580.309,Z 628.202,A -85,B 0,C 180,E1 -1929.186,E2 -1929.186} C_VEL
LIN {X 0,Y 580.279,Z 628.199,A -85,B 0,C 180,E1 -1931.768,E2 -1931.768} C_VEL
LIN {X 0,Y 580.264,Z 628.209,A -85,B 0,C 180,E1 -1934.625,E2 -1934.625} C_VEL
LIN {X 0,Y 580.28,Z 628.199,A -85,B 0,C 180,E1 -1937.294,E2 -1937.294} C_VEL
LIN {X 0,Y 580.295,Z 628.201,A -85,B 0,C 180,E1 -1940.067,E2 -1940.067} C_VEL
LIN {X 0,Y 580.3,Z 628.196,A -85,B 0,C 180,E1 -1943.064,E2 -1943.064} C_VEL
LIN {X 0,Y 580.292,Z 628.197,A -85,B 0,C 180,E1 -1945.441,E2 -1945.441} C_VEL
LIN {X 0,Y 580.304,Z 628.203,A -85,B 0,C 180,E1 -1947.968,E2 -1947.968} C_VEL
LIN {X 0,Y 580.301,Z 628.195,A -85,B 0,C 180,E1 -1950.689,E2 -1950.689} C_VEL
LIN {X 0,Y 580.323,Z 628.201,A -85,B 0,C 180,E1 -1953.658,E2 -1953.658} C_VEL
LIN {X 0,Y 580.277,Z 628.198,A -85,B 0,C 180,E1 -1956.442,E2 -1956.442} C_VEL
LIN {X 0,Y 580.28,Z 628.206,A -85,B 0,C 180,E1 -1959.437,E2 -1959.437} C_VEL
LIN {X 0,Y 580.277,Z 628.201,A -85,B 0,C 180,E1 -1961.645,E2 -1961.645} C_VEL
LIN {X 0,Y 580.275,Z 628.199,A -85,B 0,C 180,E1 -1963.825,E2 -1963.825} C_VEL
LIN {X 0,Y 580.322,Z 628.193,A -85,B 0,C 180,E1 -1965.983,E2 -1965.983} C_VEL
LIN {X 0,Y 580.327,Z 628.201,A -85,B 0,C 180,E1 -1968.827,E2 -1968.827} C_VEL
LIN {X 0,Y 580.332,Z 628.192,A -85,B 0,C 180,E1 -1971.644,E2 -1971.644} C_VEL
LIN {X 0,Y 580.317,Z 628.202,A -85,B 0,C 180,E1 -1974.44,E2 -1974.44} C_VEL
LIN {X 0,Y 580.342,Z 628.191,A -85,B 0,C 180,E1 -1977.223,E2 -1977.223} C_VEL
LIN {X 0,Y 580.347,Z 628.196,A -85,B 0,C 180,E1 -1980,E2 -1980} C_VEL
LIN {X 0,Y 580.342,Z 628.193,A -85,B 0,C 180,E1 -1982.776,E2 -1982.776} C_VEL
LIN {X 0,Y 580.359,Z 628.296,A -85,B 0,C 180,E1 -1985.254,E2 -1985.254} C_VEL
LIN {X 0,Y 580.596,Z 637.284,A -85,B 0,C 180,E1 -1987.302,E2 -1987.302} C_VEL
LIN {X 0,Y 580.783,Z 647.97,A -85,B 0,C 180,E1 -1989.754,E2 -1989.754} C_VEL
LIN {X 0,Y 580.721,Z 657.747,A -85,B 0,C 180,E1 -1992.227,E2 -1992.227} C_VEL
LIN {X 0,Y 580.583,Z 670.439,A -85,B 0,C 180,E1 -1995.445,E2 -1995.445} C_VEL
LIN {X 0,Y 580.473,Z 682.181,A -85,B 0,C 180,E1 -1998.348,E2 -1998.348} C_VEL
LIN {X 0,Y 580.427,Z 689.456,A -85,B 0,C 180,E1 -2000.117,E2 -2000.117} C_VEL
LIN {X 0,Y 579.761,Z 691.764,A -85,B 0,C 180,E1 -2000.65,E2 -2000.65} C_VEL
LIN {X 0,Y 573.945,Z 699.723,A -85,B 0,C 180,E1 -2002.366,E2 -2002.366} C_VEL
LIN {X 0,Y 573.289,Z 702.058,A -85,B 0,C 180,E1 -2002.907,E2 -2002.907} C_VEL
LIN {X 0,Y 573.23,Z 712.535,A -85,B 0,C 180,E1 -2005.411,E2 -2005.411} C_VEL
LIN {X 0,Y 573.126,Z 724.467,A -85,B 0,C 180,E1 -2008.226,E2 -2008.226} C_VEL
LIN {X 0,Y 573.108,Z 725.665,A -85,B 0,C 180,E1 -2008.507,E2 -2008.507} C_VEL
LIN {X 0,Y 573.852,Z 732.114,A -85,B 0,C 180,E1 -2008.643,E2 -2008.643} C_VEL
LIN {X 0,Y 573.788,Z 745.176,A -85,B 0,C 180,E1 -2008.972,E2 -2008.972} C_VEL
LIN {X 0,Y 573.661,Z 757.177,A -85,B 0,C 180,E1 -2009.413,E2 -2009.413} C_VEL
LIN {X 0,Y 573.532,Z 768.667,A -85,B 0,C 180,E1 -2009.975,E2 -2009.975} C_VEL
LIN {X 0,Y 573.426,Z 780.821,A -85,B 0,C 180,E1 -2010.743,E2 -2010.743} C_VEL
LIN {X 0,Y 573.307,Z 791.603,A -85,B 0,C 180,E1 -2011.605,E2 -2011.605} C_VEL
LIN {X 0,Y 573.203,Z 800.922,A -85,B 0,C 180,E1 -2012.53,E2 -2012.53} C_VEL
LIN {X 0,Y 573.137,Z 808.962,A -85,B 0,C 180,E1 -2013.506,E2 -2013.506} C_VEL
LIN {X 0,Y 573.09,Z 815.918,A -85,B 0,C 180,E1 -2014.544,E2 -2014.544} C_VEL
LIN {X 0,Y 573.051,Z 821.482,A -85,B 0,C 180,E1 -2015.574,E2 -2015.574} C_VEL
LIN {X 0,Y 573.021,Z 825.488,A -85,B 0,C 180,E1 -2016.501,E2 -2016.501} C_VEL
LIN {X 0,Y 572.985,Z 828.729,A -85,B 0,C 180,E1 -2017.453,E2 -2017.453} C_VEL
LIN {X 0,Y 572.949,Z 831.824,A -85,B 0,C 180,E1 -2018.725,E2 -2018.725} C_VEL
LIN {X 0,Y 572.93,Z 833.177,A -85,B 0,C 180,E1 -2019.633,E2 -2019.633} C_VEL
LIN {X 0,Y 572.933,Z 833.897,A -85,B 0,C 180,E1 -2020.552,E2 -2020.552} C_VEL
LIN {X 0,Y 572.96,Z 833.89,A -85,B 0,C 180,E1 -2021.564,E2 -2021.564} C_VEL
LIN {X 0,Y 572.955,Z 833.005,A -85,B 0,C 180,E1 -2022.611,E2 -2022.611} C_VEL
LIN {X 0,Y 572.934,Z 831.271,A -85,B 0,C 180,E1 -2023.637,E2 -2023.637} C_VEL
LIN {X 0,Y 572.98,Z 828.688,A -85,B 0,C 180,E1 -2024.651,E2 -2024.651} C_VEL
LIN {X 0,Y 573.003,Z 825.265,A -85,B 0,C 180,E1 -2025.645,E2 -2025.645} C_VEL
LIN {X 0,Y 573.055,Z 819.914,A -85,B 0,C 180,E1 -2026.826,E2 -2026.826} C_VEL
LIN {X 0,Y 573.086,Z 812.863,A -85,B 0,C 180,E1 -2028.031,E2 -2028.031} C_VEL
LIN {X 0,Y 573.16,Z 805.7,A -85,B 0,C 180,E1 -2029.005,E2 -2029.005} C_VEL
LIN {X 0,Y 573.245,Z 796.214,A -85,B 0,C 180,E1 -2030.051,E2 -2030.051} C_VEL
LIN {X 0,Y 573.354,Z 785.835,A -85,B 0,C 180,E1 -2030.97,E2 -2030.97} C_VEL
LIN {X 0,Y 573.483,Z 775.276,A -85,B 0,C 180,E1 -2031.721,E2 -2031.721} C_VEL
LIN {X 0,Y 573.557,Z 763.776,A -85,B 0,C 180,E1 -2032.373,E2 -2032.373} C_VEL
LIN {X 0,Y 573.749,Z 750.91,A -85,B 0,C 180,E1 -2032.924,E2 -2032.924} C_VEL
LIN {X 0,Y 573.839,Z 738.099,A -85,B 0,C 180,E1 -2033.314,E2 -2033.314} C_VEL
LIN {X 0,Y 573.732,Z 729.545,A -85,B 0,C 180,E1 -2033.497,E2 -2033.497} C_VEL
LIN {X 0,Y 573.135,Z 725.634,A -85,B 0,C 180,E1 -2033.59,E2 -2033.59} C_VEL
LIN {X 0,Y 573.179,Z 713.241,A -85,B 0,C 180,E1 -2036.513,E2 -2036.513} C_VEL
LIN {X 0,Y 573.268,Z 702.357,A -85,B 0,C 180,E1 -2039.111,E2 -2039.111} C_VEL
LIN {X 0,Y 573.366,Z 691.537,A -85,B 0,C 180,E1 -2041.733,E2 -2041.733} C_VEL
LIN {X 0,Y 573.504,Z 681.457,A -85,B 0,C 180,E1 -2044.213,E2 -2044.213} C_VEL
LIN {X 0,Y 573.599,Z 670.687,A -85,B 0,C 180,E1 -2046.917,E2 -2046.917} C_VEL
LIN {X 0,Y 573.71,Z 660.36,A -85,B 0,C 180,E1 -2049.567,E2 -2049.567} C_VEL
LIN {X 0,Y 573.746,Z 652.945,A -85,B 0,C 180,E1 -2051.429,E2 -2051.429} C_VEL
LIN {X 0,Y 573.763,Z 642.504,A -85,B 0,C 180,E1 -2054.003,E2 -2054.003} C_VEL
LIN {X 0,Y 573.645,Z 632.116,A -85,B 0,C 180,E1 -2056.54,E2 -2056.54} C_VEL
LIN {X 0,Y 573.273,Z 629.08,A -85,B 0,C 180,E1 -2057.342,E2 -2057.342} C_VEL
LIN {X 0,Y 573.234,Z 629.085,A -85,B 0,C 180,E1 -2060.117,E2 -2060.117} C_VEL
LIN {X 0,Y 573.282,Z 629.075,A -85,B 0,C 180,E1 -2062.25,E2 -2062.25} C_VEL
LIN {X 0,Y 573.312,Z 629.073,A -85,B 0,C 180,E1 -2065.078,E2 -2065.078} C_VEL
LIN {X 0,Y 573.315,Z 629.073,A -85,B 0,C 180,E1 -2067.893,E2 -2067.893} C_VEL
LIN {X 0,Y 573.338,Z 629.072,A -85,B 0,C 180,E1 -2070.703,E2 -2070.703} C_VEL
LIN {X 0,Y 573.242,Z 629.082,A -85,B 0,C 180,E1 -2073.515,E2 -2073.515} C_VEL
LIN {X 0,Y 573.289,Z 629.074,A -85,B 0,C 180,E1 -2075.629,E2 -2075.629} C_VEL
LIN {X 0,Y 573.293,Z 629.075,A -85,B 0,C 180,E1 -2078.46,E2 -2078.46} C_VEL
LIN {X 0,Y 573.275,Z 629.079,A -85,B 0,C 180,E1 -2081.312,E2 -2081.312} C_VEL
LIN {X 0,Y 573.277,Z 629.078,A -85,B 0,C 180,E1 -2084.193,E2 -2084.193} C_VEL
LIN {X 0,Y 573.263,Z 629.078,A -85,B 0,C 180,E1 -2087.112,E2 -2087.112} C_VEL
LIN {X 0,Y 573.245,Z 629.08,A -85,B 0,C 180,E1 -2090.077,E2 -2090.077} C_VEL
LIN {X 0,Y 573.24,Z 629.081,A -85,B 0,C 180,E1 -2092.338,E2 -2092.338} C_VEL
LIN {X 0,Y 573.255,Z 629.079,A -85,B 0,C 180,E1 -2095.41,E2 -2095.41} C_VEL
LIN {X 0,Y 573.284,Z 629.079,A -85,B 0,C 180,E1 -2096.091,E2 -2096.091} C_VEL
LIN {X 0,Y 573.737,Z 632.291,A -85,B 0,C 180,E1 -2096.216,E2 -2096.216} C_VEL
LIN {X 0,Y 573.623,Z 645.001,A -85,B 0,C 180,E1 -2096.782,E2 -2096.782} C_VEL
LIN {X 0,Y 573.521,Z 655.036,A -85,B 0,C 180,E1 -2097.357,E2 -2097.357} C_VEL
LIN {X 0,Y 573.406,Z 664.97,A -85,B 0,C 180,E1 -2098.058,E2 -2098.058} C_VEL
LIN {X 0,Y 573.283,Z 674.331,A -85,B 0,C 180,E1 -2098.863,E2 -2098.863} C_VEL
LIN {X 0,Y 573.162,Z 683.325,A -85,B 0,C 180,E1 -2099.803,E2 -2099.803} C_VEL
LIN {X 0,Y 573.121,Z 692.458,A -85,B 0,C 180,E1 -2101,E2 -2101} C_VEL
LIN {X 0,Y 573.085,Z 697.552,A -85,B 0,C 180,E1 -2101.825,E2 -2101.825} C_VEL
LIN {X 0,Y 572.995,Z 703.71,A -85,B 0,C 180,E1 -2103.071,E2 -2103.071} C_VEL
LIN {X 0,Y 572.986,Z 708.383,A -85,B 0,C 180,E1 -2104.348,E2 -2104.348} C_VEL
LIN {X 0,Y 572.953,Z 710.707,A -85,B 0,C 180,E1 -2105.206,E2 -2105.206} C_VEL
LIN {X 0,Y 572.922,Z 712.421,A -85,B 0,C 180,E1 -2106.073,E2 -2106.073} C_VEL
LIN {X 0,Y 572.927,Z 713.641,A -85,B 0,C 180,E1 -2107.123,E2 -2107.123} C_VEL
LIN {X 0,Y 572.928,Z 713.956,A -85,B 0,C 180,E1 -2108.272,E2 -2108.272} C_VEL
LIN {X 0,Y 572.925,Z 712.942,A -85,B 0,C 180,E1 -2109.634,E2 -2109.634} C_VEL
LIN {X 0,Y 572.938,Z 710.418,A -85,B 0,C 180,E1 -2111.016,E2 -2111.016} C_VEL
LIN {X 0,Y 573.014,Z 706.132,A -85,B 0,C 180,E1 -2112.421,E2 -2112.421} C_VEL
LIN {X 0,Y 573.005,Z 700.804,A -85,B 0,C 180,E1 -2113.644,E2 -2113.644} C_VEL
LIN {X 0,Y 573.069,Z 695.175,A -85,B 0,C 180,E1 -2114.659,E2 -2114.659} C_VEL
LIN {X 0,Y 573.129,Z 688.369,A -85,B 0,C 180,E1 -2115.656,E2 -2115.656} C_VEL
